    CONST robtarget Target_2550_2:=[[144.47,108.876,3],[0.69636424,0.122787804,0.122787804,-0.69636424],[-1,0,-1,1],[9E+09,9E+09,9E+09,9E+09,9E+09,9E+09]];
    CONST robtarget Target_2560_2:=[[144.866,108.509,3],[0.69636424,0.122787804,0.122787804,-0.69636424],[-1,0,-1,1],[9E+09,9E+09,9E+09,9E+09,9E+09,9E+09]];
    CONST robtarget Target_2570_2:=[[148.292,108.45,3],[0.69636424,0.122787804,0.122787804,-0.69636424],[-1,0,-1,1],[9E+09,9E+09,9E+09,9E+09,9E+09,9E+09]];
    CONST robtarget Target_2580_2:=[[149.079,109.372,3],[0.69636424,0.122787804,0.122787804,-0.69636424],[-1,0,-1,1],[9E+09,9E+09,9E+09,9E+09,9E+09,9E+09]];
    CONST robtarget Target_2590_2:=[[149.459,109.996,3],[0.69636424,0.122787804,0.122787804,-0.69636424],[-1,0,-1,1],[9E+09,9E+09,9E+09,9E+09,9E+09,9E+09]];
    CONST robtarget Target_2600_2:=[[149.804,110.629,3],[0.69636424,0.122787804,0.122787804,-0.69636424],[-1,0,-1,1],[9E+09,9E+09,9E+09,9E+09,9E+09,9E+09]];
    CONST robtarget Target_2610_2:=[[150.164,111.446,3],[0.69636424,0.122787804,0.122787804,-0.69636424],[-1,0,-1,1],[9E+09,9E+09,9E+09,9E+09,9E+09,9E+09]];
    CONST robtarget Target_2620_2:=[[150.582,112.397,3],[0.69636424,0.122787804,0.122787804,-0.69636424],[-1,0,-1,1],[9E+09,9E+09,9E+09,9E+09,9E+09,9E+09]];
    CONST robtarget Target_2630_2:=[[151.11,114.532,3],[0.69636424,0.122787804,0.122787804,-0.69636424],[-1,0,-1,1],[9E+09,9E+09,9E+09,9E+09,9E+09,9E+09]];
    CONST robtarget Target_2640_2:=[[151.258,118.351,3],[0.69636424,0.122787804,0.122787804,-0.69636424],[-1,0,-1,1],[9E+09,9E+09,9E+09,9E+09,9E+09,9E+09]];
    CONST robtarget Target_2650_2:=[[151.149,123.493,3],[0.69636424,0.122787804,0.122787804,-0.69636424],[-1,0,-1,1],[9E+09,9E+09,9E+09,9E+09,9E+09,9E+09]];
    CONST robtarget Target_2660_2:=[[150.509,124.998,3],[0.69636424,0.122787804,0.122787804,-0.69636424],[-1,0,-1,1],[9E+09,9E+09,9E+09,9E+09,9E+09,9E+09]];
    CONST robtarget Target_2670_2:=[[150.189,126.067,3],[0.69636424,0.122787804,0.122787804,-0.69636424],[-1,0,-1,1],[9E+09,9E+09,9E+09,9E+09,9E+09,9E+09]];
    CONST robtarget Target_2690_2:=[[149.435,127.495,3],[0.69636424,0.122787804,0.122787804,-0.69636424],[-1,0,-1,1],[9E+09,9E+09,9E+09,9E+09,9E+09,9E+09]];
    CONST robtarget Target_2700_2:=[[149.028,128.307,3],[0.69636424,0.122787804,0.122787804,-0.69636424],[-1,0,-1,1],[9E+09,9E+09,9E+09,9E+09,9E+09,9E+09]];
    CONST robtarget Target_2710_2:=[[148.353,128.811,3],[0.69636424,0.122787804,0.122787804,-0.69636424],[-1,0,-1,1],[9E+09,9E+09,9E+09,9E+09,9E+09,9E+09]];
    CONST robtarget Target_2720_2:=[[147.544,129.27,3],[0.69636424,0.122787804,0.122787804,-0.69636424],[-1,0,-1,1],[9E+09,9E+09,9E+09,9E+09,9E+09,9E+09]];
    CONST robtarget Target_2730_2:=[[146.677,129.693,3],[0.69636424,0.122787804,0.122787804,-0.69636424],[-1,0,-1,1],[9E+09,9E+09,9E+09,9E+09,9E+09,9E+09]];
    CONST robtarget Target_2740_2:=[[144.048,129.755,3],[0.69636424,0.122787804,0.122787804,-0.69636424],[-1,0,-1,1],[9E+09,9E+09,9E+09,9E+09,9E+09,9E+09]];
    CONST robtarget Target_2750_2:=[[141.627,127.645,3],[0.69636424,0.122787804,0.122787804,-0.69636424],[-1,0,-1,1],[9E+09,9E+09,9E+09,9E+09,9E+09,9E+09]];
    CONST robtarget Target_2760_2:=[[171.446,116.13,-27],[0.69636424,0.122787804,0.122787804,-0.69636424],[-1,0,-1,1],[9E+09,9E+09,9E+09,9E+09,9E+09,9E+09]];
    CONST robtarget Target_2770_2:=[[171.446,116.145,3],[0.69636424,0.122787804,0.122787804,-0.69636424],[-1,0,-1,1],[9E+09,9E+09,9E+09,9E+09,9E+09,9E+09]];
    CONST robtarget Target_2780_2:=[[171.382,110.454,3],[0.69636424,0.122787804,0.122787804,-0.69636424],[-1,0,-1,1],[9E+09,9E+09,9E+09,9E+09,9E+09,9E+09]];
    CONST robtarget Target_2790_2:=[[172.421,109.424,3],[0.69636424,0.122787804,0.122787804,-0.69636424],[-1,0,-1,1],[9E+09,9E+09,9E+09,9E+09,9E+09,9E+09]];
    CONST robtarget Target_2800_2:=[[173.527,108.448,3],[0.69636424,0.122787804,0.122787804,-0.69636424],[-1,0,-1,1],[9E+09,9E+09,9E+09,9E+09,9E+09,9E+09]];
    CONST robtarget Target_2810_2:=[[174.583,107.985,3],[0.69636424,0.122787804,0.122787804,-0.69636424],[-1,0,-1,1],[9E+09,9E+09,9E+09,9E+09,9E+09,9E+09]];
    CONST robtarget Target_2820_2:=[[175.225,107.505,3],[0.69636424,0.122787804,0.122787804,-0.69636424],[-1,0,-1,1],[9E+09,9E+09,9E+09,9E+09,9E+09,9E+09]];
    CONST robtarget Target_2830_2:=[[178.189,107.549,3],[0.69636424,0.122787804,0.122787804,-0.69636424],[-1,0,-1,1],[9E+09,9E+09,9E+09,9E+09,9E+09,9E+09]];
    CONST robtarget Target_2840_2:=[[178.951,108.484,3],[0.69636424,0.122787804,0.122787804,-0.69636424],[-1,0,-1,1],[9E+09,9E+09,9E+09,9E+09,9E+09,9E+09]];
    CONST robtarget Target_2850_2:=[[179.322,108.956,3],[0.69636424,0.122787804,0.122787804,-0.69636424],[-1,0,-1,1],[9E+09,9E+09,9E+09,9E+09,9E+09,9E+09]];
    CONST robtarget Target_2860_2:=[[179.662,109.677,3],[0.69636424,0.122787804,0.122787804,-0.69636424],[-1,0,-1,1],[9E+09,9E+09,9E+09,9E+09,9E+09,9E+09]];
    CONST robtarget Target_2870_2:=[[179.673,112.896,3],[0.69636424,0.122787804,0.122787804,-0.69636424],[-1,0,-1,1],[9E+09,9E+09,9E+09,9E+09,9E+09,9E+09]];
    CONST robtarget Target_2880_2:=[[178.94,113.73,3],[0.69636424,0.122787804,0.122787804,-0.69636424],[-1,0,-1,1],[9E+09,9E+09,9E+09,9E+09,9E+09,9E+09]];
    CONST robtarget Target_2890_2:=[[177.839,114.708,3],[0.69636424,0.122787804,0.122787804,-0.69636424],[-1,0,-1,1],[9E+09,9E+09,9E+09,9E+09,9E+09,9E+09]];
    CONST robtarget Target_2900_2:=[[175.361,115.711,3],[0.69636424,0.122787804,0.122787804,-0.69636424],[-1,0,-1,1],[9E+09,9E+09,9E+09,9E+09,9E+09,9E+09]];
    CONST robtarget Target_2910_2:=[[174.498,116.176,3],[0.69636424,0.122787804,0.122787804,-0.69636424],[-1,0,-1,1],[9E+09,9E+09,9E+09,9E+09,9E+09,9E+09]];
    CONST robtarget Target_2920_2:=[[207.225,82.129060431,2.819077862],[0.704416026,0.061628416,0.061628416,-0.704416026],[-1,0,-1,1],[9E+09,9E+09,9E+09,9E+09,9E+09,9E+09]];
    CONST robtarget Target_2920_up_2:=[[207.225,82.129060431,-27.180922138],[0.704416026,0.061628416,0.061628416,-0.704416026],[-1,0,-1,1],[9E+09,9E+09,9E+09,9E+09,9E+09,9E+09]];
    CONST robtarget Target_2930_2:=[[189.302,82.034060431,2.819077862],[0.704416026,0.061628416,0.061628416,-0.704416026],[-1,0,-1,1],[9E+09,9E+09,9E+09,9E+09,9E+09,9E+09]];
    CONST robtarget Target_2940_2:=[[172.295,56.628060431,2.819077862],[0.69636424,-0.122787804,-0.122787804,-0.69636424],[-1,0,-1,1],[9E+09,9E+09,9E+09,9E+09,9E+09,9E+09]];
    CONST robtarget Target_2950_2:=[[189.448,31.520060431,2.819077862],[0.704416026,0.061628416,0.061628416,-0.704416026],[-1,0,-1,1],[9E+09,9E+09,9E+09,9E+09,9E+09,9E+09]];
    CONST robtarget Target_2960_2:=[[207.063,31.366060431,2.819077862],[0.704416026,0.061628416,0.061628416,-0.704416026],[-1,0,-1,1],[9E+09,9E+09,9E+09,9E+09,9E+09,9E+09]];
    CONST robtarget Target_2970_2:=[[198.201,73.121060431,2.819077862],[0.704416026,0.061628416,0.061628416,-0.704416026],[-1,0,-1,1],[9E+09,9E+09,9E+09,9E+09,9E+09,9E+09]];
    CONST robtarget Target_2970_up_2:=[[198.201,73.121060431,-27.180922138],[0.704416026,0.061628416,0.061628416,-0.704416026],[-1,0,-1,1],[9E+09,9E+09,9E+09,9E+09,9E+09,9E+09]];
    CONST robtarget Target_2980_2:=[[189.482,72.946060431,2.819077862],[0.704416026,0.061628416,0.061628416,-0.704416026],[-1,0,-1,1],[9E+09,9E+09,9E+09,9E+09,9E+09,9E+09]];
    CONST robtarget Target_2990_2:=[[181.283,56.738060431,2.819077862],[0.69636424,-0.122787804,-0.122787804,-0.69636424],[-1,0,-1,1],[9E+09,9E+09,9E+09,9E+09,9E+09,9E+09]];
    CONST robtarget Target_3000_2:=[[189.826,40.515060431,2.819077862],[0.704416026,0.061628416,0.061628416,-0.704416026],[-1,0,-1,1],[9E+09,9E+09,9E+09,9E+09,9E+09,9E+09]];
    CONST robtarget Target_3010_2:=[[198.134,40.185060431,2.819077862],[0.704416026,0.061628416,0.061628416,-0.704416026],[-1,0,-1,1],[9E+09,9E+09,9E+09,9E+09,9E+09,9E+09]];
    CONST robtarget Target_3030_2_2:=[[168.856,62.045020144,-29.060307379],[0.704416026,0.061628416,0.061628416,-0.704416026],[-1,0,-1,1],[9E+09,9E+09,9E+09,9E+09,9E+09,9E+09]];
    CONST robtarget Target_3030_3:=[[168.856,62.729060431,2.819077862],[0.69636424,-0.122787804,-0.122787804,-0.69636424],[-1,0,-1,1],[9E+09,9E+09,9E+09,9E+09,9E+09,9E+09]];
    CONST robtarget Target_3040_2:=[[164.492,65.336020144,0.939692621],[0.704416026,0.061628416,0.061628416,-0.704416026],[-1,0,-1,1],[9E+09,9E+09,9E+09,9E+09,9E+09,9E+09]];
    CONST robtarget Target_3050_2:=[[159.783,67.041020144,0.939692621],[0.704416026,0.061628416,0.061628416,-0.704416026],[-1,0,-1,1],[9E+09,9E+09,9E+09,9E+09,9E+09,9E+09]];
    CONST robtarget Target_3060_2:=[[154.529,67.248020144,0.939692621],[0.704416026,0.061628416,0.061628416,-0.704416026],[-1,0,-1,1],[9E+09,9E+09,9E+09,9E+09,9E+09,9E+09]];
    CONST robtarget Target_3070_2:=[[149.168,63.265020144,0.939692621],[0.704416026,0.061628416,0.061628416,-0.704416026],[-1,0,-1,1],[9E+09,9E+09,9E+09,9E+09,9E+09,9E+09]];
    CONST robtarget Target_3080_2:=[[146.594,56.470020144,0.939692621],[0.704416026,0.061628416,0.061628416,-0.704416026],[-1,0,-1,1],[9E+09,9E+09,9E+09,9E+09,9E+09,9E+09]];
    CONST robtarget Target_3090_2:=[[146.435,30.622020144,0.939692621],[0.704416026,0.061628416,0.061628416,-0.704416026],[-1,0,-1,1],[9E+09,9E+09,9E+09,9E+09,9E+09,9E+09]];
    CONST robtarget Target_3100_2:=[[151.326,30.602020144,0.939692621],[0.704416026,0.061628416,0.061628416,-0.704416026],[-1,0,-1,1],[9E+09,9E+09,9E+09,9E+09,9E+09,9E+09]];
    CONST robtarget Target_3110_2:=[[153.44,34.909020144,0.939692621],[0.704416026,0.061628416,0.061628416,-0.704416026],[-1,0,-1,1],[9E+09,9E+09,9E+09,9E+09,9E+09,9E+09]];
    CONST robtarget Target_3120_2:=[[156.57,31.843020144,0.939692621],[0.704416026,0.061628416,0.061628416,-0.704416026],[-1,0,-1,1],[9E+09,9E+09,9E+09,9E+09,9E+09,9E+09]];
    CONST robtarget Target_3130_2:=[[160.302,30.191020144,0.939692621],[0.704416026,0.061628416,0.061628416,-0.704416026],[-1,0,-1,1],[9E+09,9E+09,9E+09,9E+09,9E+09,9E+09]];
    CONST robtarget Target_3140_2:=[[163.825,30.168020144,0.939692621],[0.704416026,0.061628416,0.061628416,-0.704416026],[-1,0,-1,1],[9E+09,9E+09,9E+09,9E+09,9E+09,9E+09]];
    CONST robtarget Target_3150_2:=[[167.12,31.969020144,0.939692621],[0.704416026,0.061628416,0.061628416,-0.704416026],[-1,0,-1,1],[9E+09,9E+09,9E+09,9E+09,9E+09,9E+09]];
    CONST robtarget Target_3160_2:=[[169.87,36.987020144,0.939692621],[0.704416026,0.061628416,0.061628416,-0.704416026],[-1,0,-1,1],[9E+09,9E+09,9E+09,9E+09,9E+09,9E+09]];
    CONST robtarget Target_3170_2:=[[170.005,41.186020144,0.939692621],[0.704416026,0.061628416,0.061628416,-0.704416026],[-1,0,-1,1],[9E+09,9E+09,9E+09,9E+09,9E+09,9E+09]];
    CONST robtarget Target_3180_2:=[[166.518,48.057020144,0.939692621],[0.704416026,0.061628416,0.061628416,-0.704416026],[-1,0,-1,1],[9E+09,9E+09,9E+09,9E+09,9E+09,9E+09]];
    CONST robtarget Target_3190_2:=[[159.562,51.317020144,0.939692621],[0.704416026,0.061628416,0.061628416,-0.704416026],[-1,0,-1,1],[9E+09,9E+09,9E+09,9E+09,9E+09,9E+09]];
    CONST robtarget Target_3200_2:=[[154.356,51.836020144,0.939692621],[0.704416026,0.061628416,0.061628416,-0.704416026],[-1,0,-1,1],[9E+09,9E+09,9E+09,9E+09,9E+09,9E+09]];
    CONST robtarget Target_3210_2:=[[154.402,56.254020144,0.939692621],[0.704416026,0.061628416,0.061628416,-0.704416026],[-1,0,-1,1],[9E+09,9E+09,9E+09,9E+09,9E+09,9E+09]];
    CONST robtarget Target_3220_2:=[[156.646,59.021020144,0.939692621],[0.704416026,0.061628416,0.061628416,-0.704416026],[-1,0,-1,1],[9E+09,9E+09,9E+09,9E+09,9E+09,9E+09]];
    CONST robtarget Target_3230_2:=[[159.999,59.059020144,0.939692621],[0.704416026,0.061628416,0.061628416,-0.704416026],[-1,0,-1,1],[9E+09,9E+09,9E+09,9E+09,9E+09,9E+09]];
    CONST robtarget Target_3240_2:=[[163.724,56.946020144,0.939692621],[0.704416026,0.061628416,0.061628416,-0.704416026],[-1,0,-1,1],[9E+09,9E+09,9E+09,9E+09,9E+09,9E+09]];
    CONST robtarget Target_3250_2:=[[166.309,56.964020144,0.939692621],[0.704416026,0.061628416,0.061628416,-0.704416026],[-1,0,-1,1],[9E+09,9E+09,9E+09,9E+09,9E+09,9E+09]];
    CONST robtarget Target_3260_2_2:=[[154.254,45.587020144,-29.060307379],[0.704416026,0.061628416,0.061628416,-0.704416026],[-1,0,-1,1],[9E+09,9E+09,9E+09,9E+09,9E+09,9E+09]];
    CONST robtarget Target_3260_3:=[[154.254,45.587020144,0.939692621],[0.69636424,-0.122787804,-0.122787804,-0.69636424],[-1,0,-1,1],[9E+09,9E+09,9E+09,9E+09,9E+09,9E+09]];
    CONST robtarget Target_3270_2:=[[154.243,40.170020144,0.939692621],[0.704416026,0.061628416,0.061628416,-0.704416026],[-1,0,-1,1],[9E+09,9E+09,9E+09,9E+09,9E+09,9E+09]];
    CONST robtarget Target_3280_2:=[[155.887,38.274020144,0.939692621],[0.704416026,0.061628416,0.061628416,-0.704416026],[-1,0,-1,1],[9E+09,9E+09,9E+09,9E+09,9E+09,9E+09]];
    CONST robtarget Target_3290_2:=[[157.675,37.336020144,0.939692621],[0.704416026,0.061628416,0.061628416,-0.704416026],[-1,0,-1,1],[9E+09,9E+09,9E+09,9E+09,9E+09,9E+09]];
    CONST robtarget Target_3300_2:=[[160.603,37.207020144,0.939692621],[0.704416026,0.061628416,0.061628416,-0.704416026],[-1,0,-1,1],[9E+09,9E+09,9E+09,9E+09,9E+09,9E+09]];
    CONST robtarget Target_3310_2:=[[162.533,39.193020144,0.939692621],[0.704416026,0.061628416,0.061628416,-0.704416026],[-1,0,-1,1],[9E+09,9E+09,9E+09,9E+09,9E+09,9E+09]];
    CONST robtarget Target_3320_2:=[[162.426,41.941020144,0.939692621],[0.704416026,0.061628416,0.061628416,-0.704416026],[-1,0,-1,1],[9E+09,9E+09,9E+09,9E+09,9E+09,9E+09]];
    CONST robtarget Target_3330_2:=[[160.229,44.430020144,0.939692621],[0.704416026,0.061628416,0.061628416,-0.704416026],[-1,0,-1,1],[9E+09,9E+09,9E+09,9E+09,9E+09,9E+09]];
    CONST robtarget Target_3340_2:=[[157.734,45.576020144,0.939692621],[0.704416026,0.061628416,0.061628416,-0.704416026],[-1,0,-1,1],[9E+09,9E+09,9E+09,9E+09,9E+09,9E+09]];
    CONST robtarget Target_3350_2_2:=[[144.461,67.032020144,-29.060307379],[0.704416026,0.061628416,0.061628416,-0.704416026],[-1,0,-1,1],[9E+09,9E+09,9E+09,9E+09,9E+09,9E+09]];
    CONST robtarget Target_3350_3:=[[144.461,67.032020144,0.939692621],[0.69636424,-0.122787804,-0.122787804,-0.69636424],[-1,0,-1,1],[9E+09,9E+09,9E+09,9E+09,9E+09,9E+09]];
    CONST robtarget Target_3360_2:=[[136.399,66.775020144,0.939692621],[0.704416026,0.061628416,0.061628416,-0.704416026],[-1,0,-1,1],[9E+09,9E+09,9E+09,9E+09,9E+09,9E+09]];
    CONST robtarget Target_3370_2:=[[130.223,41.577020144,0.939692621],[0.704416026,0.061628416,0.061628416,-0.704416026],[-1,0,-1,1],[9E+09,9E+09,9E+09,9E+09,9E+09,9E+09]];
    CONST robtarget Target_3380_2:=[[123.937,66.551020144,0.939692621],[0.704416026,0.061628416,0.061628416,-0.704416026],[-1,0,-1,1],[9E+09,9E+09,9E+09,9E+09,9E+09,9E+09]];
    CONST robtarget Target_3390_2:=[[115.96,66.627020144,0.939692621],[0.704416026,0.061628416,0.061628416,-0.704416026],[-1,0,-1,1],[9E+09,9E+09,9E+09,9E+09,9E+09,9E+09]];
    CONST robtarget Target_3400_2:=[[126.475,30.638020144,0.939692621],[0.704416026,0.061628416,0.061628416,-0.704416026],[-1,0,-1,1],[9E+09,9E+09,9E+09,9E+09,9E+09,9E+09]];
    CONST robtarget Target_3410_2:=[[133.864,30.673020144,0.939692621],[0.704416026,0.061628416,0.061628416,-0.704416026],[-1,0,-1,1],[9E+09,9E+09,9E+09,9E+09,9E+09,9E+09]];
    CONST robtarget Target_3420_2_2:=[[112.825,66.820020144,-29.060307379],[0.704416026,0.061628416,0.061628416,-0.704416026],[-1,0,-1,1],[9E+09,9E+09,9E+09,9E+09,9E+09,9E+09]];
    CONST robtarget Target_3420_3:=[[112.825,66.820020144,0.939692621],[0.69636424,-0.122787804,-0.122787804,-0.69636424],[-1,0,-1,1],[9E+09,9E+09,9E+09,9E+09,9E+09,9E+09]];
    CONST robtarget Target_3430_2:=[[104.746,66.822020144,0.939692621],[0.704416026,0.061628416,0.061628416,-0.704416026],[-1,0,-1,1],[9E+09,9E+09,9E+09,9E+09,9E+09,9E+09]];
    CONST robtarget Target_3440_2:=[[104.632,30.482020144,0.939692621],[0.704416026,0.061628416,0.061628416,-0.704416026],[-1,0,-1,1],[9E+09,9E+09,9E+09,9E+09,9E+09,9E+09]];
    CONST robtarget Target_3450_2:=[[112.782,30.740020144,0.939692621],[0.704416026,0.061628416,0.061628416,-0.704416026],[-1,0,-1,1],[9E+09,9E+09,9E+09,9E+09,9E+09,9E+09]];
    CONST robtarget Target_3460_2_2:=[[107.732,82.799020144,-29.060307379],[0.704416026,0.061628416,0.061628416,-0.704416026],[-1,0,-1,1],[9E+09,9E+09,9E+09,9E+09,9E+09,9E+09]];
    CONST robtarget Target_3460_3:=[[107.732,82.799020144,0.939692621],[0.69636424,-0.122787804,-0.122787804,-0.69636424],[-1,0,-1,1],[9E+09,9E+09,9E+09,9E+09,9E+09,9E+09]];
    CONST robtarget Target_3470_2:=[[103.914,76.496020144,0.939692621],[0.704416026,0.061628416,0.061628416,-0.704416026],[-1,0,-1,1],[9E+09,9E+09,9E+09,9E+09,9E+09,9E+09]];
    CONST robtarget Target_3480_2:=[[107.812,70.304020144,0.939692621],[0.704416026,0.061628416,0.061628416,-0.704416026],[-1,0,-1,1],[9E+09,9E+09,9E+09,9E+09,9E+09,9E+09]];
    CONST robtarget Target_3490_2:=[[110.105,70.397020144,0.939692621],[0.704416026,0.061628416,0.061628416,-0.704416026],[-1,0,-1,1],[9E+09,9E+09,9E+09,9E+09,9E+09,9E+09]];
    CONST robtarget Target_3500_2:=[[113.61,76.180020144,0.939692621],[0.704416026,0.061628416,0.061628416,-0.704416026],[-1,0,-1,1],[9E+09,9E+09,9E+09,9E+09,9E+09,9E+09]];
    CONST robtarget Target_3510_2:=[[110.04,82.825020144,0.939692621],[0.704416026,0.061628416,0.061628416,-0.704416026],[-1,0,-1,1],[9E+09,9E+09,9E+09,9E+09,9E+09,9E+09]];
    CONST robtarget Target_3520_2_2:=[[82.277,82.761020144,-29.060307379],[0.704416026,0.061628416,0.061628416,-0.704416026],[-1,0,-1,1],[9E+09,9E+09,9E+09,9E+09,9E+09,9E+09]];
    CONST robtarget Target_3520_3:=[[82.277,82.761020144,0.939692621],[0.69636424,-0.122787804,-0.122787804,-0.69636424],[-1,0,-1,1],[9E+09,9E+09,9E+09,9E+09,9E+09,9E+09]];
    CONST robtarget Target_3530_2:=[[74.455,82.673020144,0.939692621],[0.704416026,0.061628416,0.061628416,-0.704416026],[-1,0,-1,1],[9E+09,9E+09,9E+09,9E+09,9E+09,9E+09]];
    CONST robtarget Target_3540_2:=[[74.428,30.709020144,0.939692621],[0.704416026,0.061628416,0.061628416,-0.704416026],[-1,0,-1,1],[9E+09,9E+09,9E+09,9E+09,9E+09,9E+09]];
    CONST robtarget Target_3550_2:=[[80.004,30.702020144,0.939692621],[0.704416026,0.061628416,0.061628416,-0.704416026],[-1,0,-1,1],[9E+09,9E+09,9E+09,9E+09,9E+09,9E+09]];
    CONST robtarget Target_3560_2:=[[82.07,35.013020144,0.939692621],[0.704416026,0.061628416,0.061628416,-0.704416026],[-1,0,-1,1],[9E+09,9E+09,9E+09,9E+09,9E+09,9E+09]];
    CONST robtarget Target_3570_2:=[[84.954,31.898020144,0.939692621],[0.704416026,0.061628416,0.061628416,-0.704416026],[-1,0,-1,1],[9E+09,9E+09,9E+09,9E+09,9E+09,9E+09]];
    CONST robtarget Target_3580_2:=[[88.431,30.331020144,0.939692621],[0.704416026,0.061628416,0.061628416,-0.704416026],[-1,0,-1,1],[9E+09,9E+09,9E+09,9E+09,9E+09,9E+09]];
    CONST robtarget Target_3590_2:=[[92.072,30.216020144,0.939692621],[0.704416026,0.061628416,0.061628416,-0.704416026],[-1,0,-1,1],[9E+09,9E+09,9E+09,9E+09,9E+09,9E+09]];
    CONST robtarget Target_3600_2:=[[97.435,34.873020144,0.939692621],[0.704416026,0.061628416,0.061628416,-0.704416026],[-1,0,-1,1],[9E+09,9E+09,9E+09,9E+09,9E+09,9E+09]];
    CONST robtarget Target_3610_2:=[[99.865,42.963020144,0.939692621],[0.704416026,0.061628416,0.061628416,-0.704416026],[-1,0,-1,1],[9E+09,9E+09,9E+09,9E+09,9E+09,9E+09]];
    CONST robtarget Target_3620_2:=[[100.165,49.389020144,0.939692621],[0.704416026,0.061628416,0.061628416,-0.704416026],[-1,0,-1,1],[9E+09,9E+09,9E+09,9E+09,9E+09,9E+09]];
    CONST robtarget Target_3630_2:=[[97.664,60.583020144,0.939692621],[0.704416026,0.061628416,0.061628416,-0.704416026],[-1,0,-1,1],[9E+09,9E+09,9E+09,9E+09,9E+09,9E+09]];
    CONST robtarget Target_3640_2:=[[90.704,67.178020144,0.939692621],[0.704416026,0.061628416,0.061628416,-0.704416026],[-1,0,-1,1],[9E+09,9E+09,9E+09,9E+09,9E+09,9E+09]];
    CONST robtarget Target_3650_2:=[[86.592,67.289020144,0.939692621],[0.704416026,0.061628416,0.061628416,-0.704416026],[-1,0,-1,1],[9E+09,9E+09,9E+09,9E+09,9E+09,9E+09]];
    CONST robtarget Target_3660_2:=[[82.282,64.136020144,0.939692621],[0.704416026,0.061628416,0.061628416,-0.704416026],[-1,0,-1,1],[9E+09,9E+09,9E+09,9E+09,9E+09,9E+09]];
    CONST robtarget Target_3670_2_2:=[[82.253,56.509020144,-29.060307379],[0.704416026,0.061628416,0.061628416,-0.704416026],[-1,0,-1,1],[9E+09,9E+09,9E+09,9E+09,9E+09,9E+09]];
    CONST robtarget Target_3670_3:=[[82.253,56.509020144,0.939692621],[0.69636424,-0.122787804,-0.122787804,-0.69636424],[-1,0,-1,1],[9E+09,9E+09,9E+09,9E+09,9E+09,9E+09]];
    CONST robtarget Target_3680_2:=[[82.272,41.520020144,0.939692621],[0.704416026,0.061628416,0.061628416,-0.704416026],[-1,0,-1,1],[9E+09,9E+09,9E+09,9E+09,9E+09,9E+09]];
    CONST robtarget Target_3690_2:=[[85.391,38.217020144,0.939692621],[0.704416026,0.061628416,0.061628416,-0.704416026],[-1,0,-1,1],[9E+09,9E+09,9E+09,9E+09,9E+09,9E+09]];
    CONST robtarget Target_3700_2:=[[88.811,38.071020144,0.939692621],[0.704416026,0.061628416,0.061628416,-0.704416026],[-1,0,-1,1],[9E+09,9E+09,9E+09,9E+09,9E+09,9E+09]];
    CONST robtarget Target_3710_2:=[[91.889,43.979020144,0.939692621],[0.704416026,0.061628416,0.061628416,-0.704416026],[-1,0,-1,1],[9E+09,9E+09,9E+09,9E+09,9E+09,9E+09]];
    CONST robtarget Target_3720_2:=[[92.083,51.104020144,0.939692621],[0.704416026,0.061628416,0.061628416,-0.704416026],[-1,0,-1,1],[9E+09,9E+09,9E+09,9E+09,9E+09,9E+09]];
    CONST robtarget Target_3730_2:=[[89.43,58.065020144,0.939692621],[0.704416026,0.061628416,0.061628416,-0.704416026],[-1,0,-1,1],[9E+09,9E+09,9E+09,9E+09,9E+09,9E+09]];
    CONST robtarget Target_3740_2:=[[85.526,58.965020144,0.939692621],[0.704416026,0.061628416,0.061628416,-0.704416026],[-1,0,-1,1],[9E+09,9E+09,9E+09,9E+09,9E+09,9E+09]];
    CONST robtarget Target_3750_2_2:=[[64.524,146.437020144,-29.060307379],[0.704416026,0.061628416,0.061628416,-0.704416026],[-1,0,-1,1],[9E+09,9E+09,9E+09,9E+09,9E+09,9E+09]];
    CONST robtarget Target_3750_3:=[[64.524,146.437020144,0.939692621],[0.69636424,-0.122787804,-0.122787804,-0.69636424],[-1,0,-1,1],[9E+09,9E+09,9E+09,9E+09,9E+09,9E+09]];
    CONST robtarget Target_3760_2:=[[55.549,133.666020144,0.939692621],[0.704416026,0.061628416,0.061628416,-0.704416026],[-1,0,-1,1],[9E+09,9E+09,9E+09,9E+09,9E+09,9E+09]];
    CONST robtarget Target_3770_2:=[[47.044,128.487020144,0.939692621],[0.704416026,0.061628416,0.061628416,-0.704416026],[-1,0,-1,1],[9E+09,9E+09,9E+09,9E+09,9E+09,9E+09]];
    CONST robtarget Target_3780_2:=[[37.688,111.228020144,0.939692621],[0.704416026,0.061628416,0.061628416,-0.704416026],[-1,0,-1,1],[9E+09,9E+09,9E+09,9E+09,9E+09,9E+09]];
    CONST robtarget Target_3790_2:=[[41.259,123.994020144,0.939692621],[0.704416026,0.061628416,0.061628416,-0.704416026],[-1,0,-1,1],[9E+09,9E+09,9E+09,9E+09,9E+09,9E+09]];
    CONST robtarget Target_3800_2:=[[26.923,126.980020144,0.939692621],[0.704416026,0.061628416,0.061628416,-0.704416026],[-1,0,-1,1],[9E+09,9E+09,9E+09,9E+09,9E+09,9E+09]];
    CONST robtarget Target_3810_2:=[[26.91,85.429020144,0.939692621],[0.704416026,0.061628416,0.061628416,-0.704416026],[-1,0,-1,1],[9E+09,9E+09,9E+09,9E+09,9E+09,9E+09]];
    CONST robtarget Target_3820_2:=[[31.003,81.597020144,0.939692621],[0.704416026,0.061628416,0.061628416,-0.704416026],[-1,0,-1,1],[9E+09,9E+09,9E+09,9E+09,9E+09,9E+09]];
    CONST robtarget Target_3830_2:=[[35.653,89.236020144,0.939692621],[0.704416026,0.061628416,0.061628416,-0.704416026],[-1,0,-1,1],[9E+09,9E+09,9E+09,9E+09,9E+09,9E+09]];
    CONST robtarget Target_3840_2:=[[41.161,97.045020144,0.939692621],[0.704416026,0.061628416,0.061628416,-0.704416026],[-1,0,-1,1],[9E+09,9E+09,9E+09,9E+09,9E+09,9E+09]];
    CONST robtarget Target_3850_2:=[[45.695,102.026020144,0.939692621],[0.704416026,0.061628416,0.061628416,-0.704416026],[-1,0,-1,1],[9E+09,9E+09,9E+09,9E+09,9E+09,9E+09]];
    CONST robtarget Target_3860_2:=[[52.946,106.880020144,0.939692621],[0.704416026,0.061628416,0.061628416,-0.704416026],[-1,0,-1,1],[9E+09,9E+09,9E+09,9E+09,9E+09,9E+09]];
    CONST robtarget Target_3870_2:=[[62.408,123.824020144,0.939692621],[0.704416026,0.061628416,0.061628416,-0.704416026],[-1,0,-1,1],[9E+09,9E+09,9E+09,9E+09,9E+09,9E+09]];
    CONST robtarget Target_3880_2:=[[52.276,112.163020144,0.939692621],[0.704416026,0.061628416,0.061628416,-0.704416026],[-1,0,-1,1],[9E+09,9E+09,9E+09,9E+09,9E+09,9E+09]];
    CONST robtarget Target_3890_2:=[[59.313,122.581020144,0.939692621],[0.704416026,0.061628416,0.061628416,-0.704416026],[-1,0,-1,1],[9E+09,9E+09,9E+09,9E+09,9E+09,9E+09]];
    CONST robtarget Target_3900_2:=[[63.763,135.404020144,0.939692621],[0.704416026,0.061628416,0.061628416,-0.704416026],[-1,0,-1,1],[9E+09,9E+09,9E+09,9E+09,9E+09,9E+09]];
    CONST robtarget Target_3910_2_2:=[[27.611,83.068020144,-29.060307379],[0.704416026,0.061628416,0.061628416,-0.704416026],[-1,0,-1,1],[9E+09,9E+09,9E+09,9E+09,9E+09,9E+09]];
    CONST robtarget Target_3910_3:=[[27.611,83.068020144,0.939692621],[0.69636424,-0.122787804,-0.122787804,-0.69636424],[-1,0,-1,1],[9E+09,9E+09,9E+09,9E+09,9E+09,9E+09]];
    CONST robtarget Target_3920_2:=[[24.514,80.149020144,0.939692621],[0.704416026,0.061628416,0.061628416,-0.704416026],[-1,0,-1,1],[9E+09,9E+09,9E+09,9E+09,9E+09,9E+09]];
    CONST robtarget Target_3930_2:=[[24.493,70.759020144,0.939692621],[0.704416026,0.061628416,0.061628416,-0.704416026],[-1,0,-1,1],[9E+09,9E+09,9E+09,9E+09,9E+09,9E+09]];
    CONST robtarget Target_3940_2:=[[26.846,61.477020144,0.939692621],[0.704416026,0.061628416,0.061628416,-0.704416026],[-1,0,-1,1],[9E+09,9E+09,9E+09,9E+09,9E+09,9E+09]];
    CONST robtarget Target_3950_2:=[[29.828,69.272020144,0.939692621],[0.704416026,0.061628416,0.061628416,-0.704416026],[-1,0,-1,1],[9E+09,9E+09,9E+09,9E+09,9E+09,9E+09]];
    CONST robtarget Target_3960_2:=[[30.012,78.359020144,0.939692621],[0.704416026,0.061628416,0.061628416,-0.704416026],[-1,0,-1,1],[9E+09,9E+09,9E+09,9E+09,9E+09,9E+09]];
    CONST robtarget Target_3970_2_2:=[[44.273,96.711020144,-29.060307379],[0.704416026,0.061628416,0.061628416,-0.704416026],[-1,0,-1,1],[9E+09,9E+09,9E+09,9E+09,9E+09,9E+09]];
    CONST robtarget Target_3970_3:=[[44.273,96.711020144,0.939692621],[0.69636424,-0.122787804,-0.122787804,-0.69636424],[-1,0,-1,1],[9E+09,9E+09,9E+09,9E+09,9E+09,9E+09]];
    CONST robtarget Target_3980_2:=[[43.933,86.227020144,0.939692621],[0.704416026,0.061628416,0.061628416,-0.704416026],[-1,0,-1,1],[9E+09,9E+09,9E+09,9E+09,9E+09,9E+09]];
    CONST robtarget Target_3990_2:=[[39.768,82.418020144,0.939692621],[0.704416026,0.061628416,0.061628416,-0.704416026],[-1,0,-1,1],[9E+09,9E+09,9E+09,9E+09,9E+09,9E+09]];
    CONST robtarget Target_4000_2:=[[34.596,82.452020144,0.939692621],[0.704416026,0.061628416,0.061628416,-0.704416026],[-1,0,-1,1],[9E+09,9E+09,9E+09,9E+09,9E+09,9E+09]];
    CONST robtarget Target_4010_2_2:=[[26.792,57.803020144,-29.060307379],[0.704416026,0.061628416,0.061628416,-0.704416026],[-1,0,-1,1],[9E+09,9E+09,9E+09,9E+09,9E+09,9E+09]];
    CONST robtarget Target_4010_3:=[[26.792,57.803020144,0.939692621],[0.69636424,-0.122787804,-0.122787804,-0.69636424],[-1,0,-1,1],[9E+09,9E+09,9E+09,9E+09,9E+09,9E+09]];
    CONST robtarget Target_4020_2:=[[45.072,60.926020144,0.939692621],[0.704416026,0.061628416,0.061628416,-0.704416026],[-1,0,-1,1],[9E+09,9E+09,9E+09,9E+09,9E+09,9E+09]];
    CONST robtarget Target_4030_2:=[[61.878,52.724020144,0.939692621],[0.704416026,0.061628416,0.061628416,-0.704416026],[-1,0,-1,1],[9E+09,9E+09,9E+09,9E+09,9E+09,9E+09]];
    CONST robtarget Target_4040_2:=[[59.898,63.620020144,0.939692621],[0.704416026,0.061628416,0.061628416,-0.704416026],[-1,0,-1,1],[9E+09,9E+09,9E+09,9E+09,9E+09,9E+09]];
    CONST robtarget Target_4050_2:=[[56.445,72.459020144,0.939692621],[0.704416026,0.061628416,0.061628416,-0.704416026],[-1,0,-1,1],[9E+09,9E+09,9E+09,9E+09,9E+09,9E+09]];
    CONST robtarget Target_4060_2:=[[58.835,86.000020144,0.939692621],[0.704416026,0.061628416,0.061628416,-0.704416026],[-1,0,-1,1],[9E+09,9E+09,9E+09,9E+09,9E+09,9E+09]];
    CONST robtarget Target_4070_2:=[[54.916,107.364020144,0.939692621],[0.704416026,0.061628416,0.061628416,-0.704416026],[-1,0,-1,1],[9E+09,9E+09,9E+09,9E+09,9E+09,9E+09]];
    CONST robtarget Target_4080_2:=[[49.508,100.246020144,0.939692621],[0.704416026,0.061628416,0.061628416,-0.704416026],[-1,0,-1,1],[9E+09,9E+09,9E+09,9E+09,9E+09,9E+09]];
    CONST robtarget Target_4090_2:=[[52.038,93.753020144,0.939692621],[0.704416026,0.061628416,0.061628416,-0.704416026],[-1,0,-1,1],[9E+09,9E+09,9E+09,9E+09,9E+09,9E+09]];
    CONST robtarget Target_4100_2:=[[52.392,84.414020144,0.939692621],[0.704416026,0.061628416,0.061628416,-0.704416026],[-1,0,-1,1],[9E+09,9E+09,9E+09,9E+09,9E+09,9E+09]];
    CONST robtarget Target_4110_2:=[[48.592,78.019020144,0.939692621],[0.704416026,0.061628416,0.061628416,-0.704416026],[-1,0,-1,1],[9E+09,9E+09,9E+09,9E+09,9E+09,9E+09]];
    CONST robtarget Target_4120_2:=[[44.019,73.976020144,0.939692621],[0.704416026,0.061628416,0.061628416,-0.704416026],[-1,0,-1,1],[9E+09,9E+09,9E+09,9E+09,9E+09,9E+09]];
    CONST robtarget Target_4130_2:=[[36.693,67.321020144,0.939692621],[0.704416026,0.061628416,0.061628416,-0.704416026],[-1,0,-1,1],[9E+09,9E+09,9E+09,9E+09,9E+09,9E+09]];



    PROC main()
        TPErase;
        TPWrite "Iniciando Ciclo";
        !Aqui  se reinicia todas las entradas y salidad a usar.
        Reset Conveyor_INV;
        Reset DO_01;
        Reset DO_02;
        GoHome;
        TPWrite "Porfavor presione Bot n1 para iniciar Rutina de decoracion ";
        TPWrite "Tambien, puede presionar Bot n2 para iniciar Rutina de Matenimiento ";

   WHILE TRUE DO
            IF DI_01 = 1 AND DI_02 = 0 THEN  !verificar que solo se presiono un bot n
                TPWrite "Comenzando avance de la banda";
                Set Conveyor_INV;
                WaitTime 8.7;  !cambiar este para modificar tiempo de espera entre encendido y apagado 10.2 simulaci n, 4 en real
                Reset Conveyor_INV;
                TPWrite "Banda transportadora detenida";
                TPWrite "Iniciando Decoraci n del pastel";
                Set DO_01; ! bombillo que avisa del proceso de decoraci n
                MoveAbsJ RomperSingular, v1000, z1, Soporte_final;
                Path_40;
                Path_10; ! Primero Ariadna
                TPWrite "Decoraci n ------> 34%";
                Path_20;
                TPWrite "Decoraci n ------> 67%";
                Path_30;
                TPWrite "Decoraci n ------> 100%";
                GoHome;
                WaitTime 2; !verificar este Gohome que hace.
                TPWrite "Comenzando avance de la banda";
                Set Conveyor_INV;
                WaitTime 3; ! si la caja se cae es por esto en simulaci n 3, 0.2 en real
                Reset Conveyor_INV;
                TPWrite "Banda transportadora detenida";


            ELSEIF DI_01 = 0 AND DI_02=1 THEN
                TPWrite "Rutina de Mantenimiento empezando";
                Reset DO_01; ! apagando indicador de rutina de decoraci n
                Set DO_02; ! indicador de la rutina de mantenimiento
                GoHome;
                MoveAbsJ cambio_Tool, v300, z5, Soporte_final;
                TPWrite "CUIDADO OPERARIO CERCA AL ROBOT";
                TPWrite "Presione Boton1 y Boton2 al tiempo, para continuar";
                WaitUntil DI_01=1 AND DI_02=1;
                TPWrite "Continuando Programa...";
                WaitTime 6; ! tiempo de espera para asegurarse que el operario salio.
                MoveAbsJ HOME_Origen, v300, fine, Soporte_final;
                Reset DO_02;
            ELSEIF DI_01 = 0 AND DI_02=0 THEN
                TPWrite "Esperando Instrucciones";
                ! aqui iba un Waittime pero no pienso que sea neccesario
            ENDIF
             ! revisar si es necesario otro estado
        ENDWHILE


    ENDPROC

       PROC GoHome()
        CONST num tolerancia := 0.2;
        VAR jointtarget jt;
        jt := CJointT(); ! posici n actual del robot
        IF  Abs(jt.robax.rax_1) < tolerancia AND
            Abs(jt.robax.rax_2) < tolerancia AND
            Abs(jt.robax.rax_3) < tolerancia AND
            Abs(jt.robax.rax_4) < tolerancia AND
            Abs(jt.robax.rax_5) < tolerancia AND
            Abs(jt.robax.rax_6) < tolerancia THEN
            TPWrite "Robot en home articular en 0 ";
        ELSE
            TPWrite "Yendo a Home";

            MoveAbsJ HOME_Origen, v100, fine, Soporte_final;
            TPWrite "Robot en Home";
        ENDIF
    ENDPROC

  PROC Path_10()
        MoveJ Target_minihome,v100,z5,Soporte_final\WObj:=ADwob;
        MoveJ Target_200,v100,z5,Soporte_final\WObj:=ADwob;
        MoveL Target_210,v100,z5,Soporte_final\WObj:=ADwob;
        MoveL Target_220,v100,z5,Soporte_final\WObj:=ADwob;
        MoveL Target_230,v100,z5,Soporte_final\WObj:=ADwob;
        MoveL Target_240,v100,z5,Soporte_final\WObj:=ADwob;
        MoveL Target_250,v100,z5,Soporte_final\WObj:=ADwob;
        MoveL Target_260,v100,z5,Soporte_final\WObj:=ADwob;
        MoveL Target_270,v100,z5,Soporte_final\WObj:=ADwob;
        MoveL Target_280,v100,z5,Soporte_final\WObj:=ADwob;
        MoveL Target_210,v100,z5,Soporte_final\WObj:=ADwob;
        MoveL Target_200,v100,z5,Soporte_final\WObj:=ADwob;
        MoveL Target_290,v100,z5,Soporte_final\WObj:=ADwob;
        MoveL Target_300,v100,z5,Soporte_final\WObj:=ADwob;
        MoveL Target_310,v100,z5,Soporte_final\WObj:=ADwob;
        MoveL Target_320,v100,z5,Soporte_final\WObj:=ADwob;
        MoveL Target_300,v100,z5,Soporte_final\WObj:=ADwob;
        MoveL Target_290,v100,z5,Soporte_final\WObj:=ADwob;
        MoveL Target_330,v100,z5,Soporte_final\WObj:=ADwob;
        MoveL Target_340,v100,z5,Soporte_final\WObj:=ADwob;
        MoveL Target_350,v100,z5,Soporte_final\WObj:=ADwob;
        MoveL Target_360,v100,z5,Soporte_final\WObj:=ADwob;
        MoveL Target_370,v100,z5,Soporte_final\WObj:=ADwob;
        MoveL Target_380,v100,z5,Soporte_final\WObj:=ADwob;
        MoveL Target_390,v100,z5,Soporte_final\WObj:=ADwob;
        MoveL Target_400,v100,z5,Soporte_final\WObj:=ADwob;
        MoveL Target_410,v100,z5,Soporte_final\WObj:=ADwob;
        MoveL Target_420,v100,z5,Soporte_final\WObj:=ADwob;
        MoveL Target_430,v100,z5,Soporte_final\WObj:=ADwob;
        MoveL Target_440,v100,z5,Soporte_final\WObj:=ADwob;
        MoveL Target_340,v100,z5,Soporte_final\WObj:=ADwob;
        MoveL Target_330,v100,z5,Soporte_final\WObj:=ADwob;
        MoveL Target_450,v100,z5,Soporte_final\WObj:=ADwob;
        MoveL Target_460,v100,z5,Soporte_final\WObj:=ADwob;
        MoveL Target_470,v100,z5,Soporte_final\WObj:=ADwob;
        MoveL Target_480,v100,z5,Soporte_final\WObj:=ADwob;
        MoveL Target_490,v100,z5,Soporte_final\WObj:=ADwob;
        MoveL Target_460,v100,z5,Soporte_final\WObj:=ADwob;
        MoveL Target_450,v100,z5,Soporte_final\WObj:=ADwob;
        MoveL Target_500,v100,z5,Soporte_final\WObj:=ADwob;
        MoveL Target_510,v100,z5,Soporte_final\WObj:=ADwob;
        MoveL Target_520,v100,z5,Soporte_final\WObj:=ADwob;
        MoveL Target_530,v100,z5,Soporte_final\WObj:=ADwob;
        MoveL Target_540,v100,z5,Soporte_final\WObj:=ADwob;
        MoveL Target_550,v100,z5,Soporte_final\WObj:=ADwob;
        MoveL Target_560,v100,z5,Soporte_final\WObj:=ADwob;
        MoveL Target_570,v100,z5,Soporte_final\WObj:=ADwob;
        MoveL Target_580,v100,z5,Soporte_final\WObj:=ADwob;
        MoveL Target_590,v100,z5,Soporte_final\WObj:=ADwob;
        MoveL Target_500,v100,z5,Soporte_final\WObj:=ADwob;
        MoveL Target_600,v100,z5,Soporte_final\WObj:=ADwob;
        MoveL Target_610,v100,z5,Soporte_final\WObj:=ADwob; !baja en z letra 2 a
        MoveL Target_620,v100,z5,Soporte_final\WObj:=ADwob;
        MoveL Target_630,v100,z5,Soporte_final\WObj:=ADwob;
        MoveL Target_640,v100,z5,Soporte_final\WObj:=ADwob;
        MoveL Target_650,v100,z5,Soporte_final\WObj:=ADwob;
        MoveL Target_660,v100,z5,Soporte_final\WObj:=ADwob;
        MoveL Target_670,v100,z5,Soporte_final\WObj:=ADwob;
        MoveL Target_680,v100,z5,Soporte_final\WObj:=ADwob;
        MoveL Target_690,v100,z5,Soporte_final\WObj:=ADwob;
        MoveL Target_700,v100,z5,Soporte_final\WObj:=ADwob;
        MoveL Target_710,v100,z5,Soporte_final\WObj:=ADwob;
        MoveL Target_720,v100,z5,Soporte_final\WObj:=ADwob;
        MoveL Target_730,v100,z5,Soporte_final\WObj:=ADwob;
        MoveL Target_740,v100,z5,Soporte_final\WObj:=ADwob;
        MoveL Target_750,v100,z5,Soporte_final\WObj:=ADwob;
        MoveL Target_760,v100,z5,Soporte_final\WObj:=ADwob;
        MoveL Target_770,v100,z5,Soporte_final\WObj:=ADwob;
        MoveL Target_780,v100,z5,Soporte_final\WObj:=ADwob;
        MoveL Target_790,v100,z5,Soporte_final\WObj:=ADwob;
        MoveL Target_800,v100,z5,Soporte_final\WObj:=ADwob;
        MoveL Target_810,v100,z5,Soporte_final\WObj:=ADwob;
        MoveL Target_820,v100,z5,Soporte_final\WObj:=ADwob;
        MoveL Target_830,v100,z5,Soporte_final\WObj:=ADwob;
        MoveL Target_840,v100,z5,Soporte_final\WObj:=ADwob;
        MoveL Target_850,v100,z5,Soporte_final\WObj:=ADwob;
        MoveL Target_860,v100,z5,Soporte_final\WObj:=ADwob;
        MoveL Target_870,v100,z5,Soporte_final\WObj:=ADwob;
        MoveL Target_880,v100,z5,Soporte_final\WObj:=ADwob;
        MoveL Target_890,v100,z5,Soporte_final\WObj:=ADwob;
        MoveL Target_900,v100,z5,Soporte_final\WObj:=ADwob;
        MoveL Target_610,v100,z5,Soporte_final\WObj:=ADwob; !une las cosas en a
        MoveL Target_600,v100,z5,Soporte_final\WObj:=ADwob;
        MoveL Target_910,v100,z5,Soporte_final\WObj:=ADwob;
        MoveL Target_920,v100,z5,Soporte_final\WObj:=ADwob;
        MoveL Target_930,v100,z5,Soporte_final\WObj:=ADwob;
        MoveL Target_940,v100,z5,Soporte_final\WObj:=ADwob;
        MoveL Target_950,v100,z5,Soporte_final\WObj:=ADwob;
        MoveL Target_960,v100,z5,Soporte_final\WObj:=ADwob;
        MoveL Target_970,v100,z5,Soporte_final\WObj:=ADwob;
        MoveL Target_980,v100,z5,Soporte_final\WObj:=ADwob;
        MoveL Target_990,v100,z5,Soporte_final\WObj:=ADwob;
        MoveL Target_1000,v100,z5,Soporte_final\WObj:=ADwob;
        MoveL Target_1010,v100,z5,Soporte_final\WObj:=ADwob;
        MoveL Target_1020,v100,z5,Soporte_final\WObj:=ADwob;
        MoveL Target_1030,v100,z5,Soporte_final\WObj:=ADwob;
        MoveL Target_1040,v100,z5,Soporte_final\WObj:=ADwob;
        MoveL Target_1050,v100,z5,Soporte_final\WObj:=ADwob;
        MoveL Target_1060,v100,z5,Soporte_final\WObj:=ADwob;
        MoveL Target_1070,v100,z5,Soporte_final\WObj:=ADwob;
        MoveL Target_1080,v100,z5,Soporte_final\WObj:=ADwob;
        MoveL Target_1090,v100,z5,Soporte_final\WObj:=ADwob;
        MoveL Target_1100,v100,z5,Soporte_final\WObj:=ADwob;
        MoveL Target_920,v100,z5,Soporte_final\WObj:=ADwob;
        MoveL Target_910,v100,z5,Soporte_final\WObj:=ADwob;
        MoveL Target_1110,v100,z5,Soporte_final\WObj:=ADwob;
        MoveL Target_1120,v100,z5,Soporte_final\WObj:=ADwob;
        MoveL Target_1130,v100,z5,Soporte_final\WObj:=ADwob;
        MoveL Target_1140,v100,z5,Soporte_final\WObj:=ADwob;
        MoveL Target_1150,v100,z5,Soporte_final\WObj:=ADwob;
        MoveL Target_1160,v100,z5,Soporte_final\WObj:=ADwob;
        MoveL Target_1170,v100,z5,Soporte_final\WObj:=ADwob;
        MoveL Target_1180,v100,z5,Soporte_final\WObj:=ADwob;
        MoveL Target_1190,v100,z5,Soporte_final\WObj:=ADwob;
        MoveL Target_1200,v100,z5,Soporte_final\WObj:=ADwob;
        MoveL Target_1210,v100,z5,Soporte_final\WObj:=ADwob;
        MoveL Target_1220,v100,z5,Soporte_final\WObj:=ADwob;
        MoveL Target_1230,v100,z5,Soporte_final\WObj:=ADwob;
        MoveL Target_1240,v100,z5,Soporte_final\WObj:=ADwob;
        MoveL Target_1250,v100,z5,Soporte_final\WObj:=ADwob;
        MoveL Target_1260,v100,z5,Soporte_final\WObj:=ADwob;
        MoveL Target_1270,v100,z5,Soporte_final\WObj:=ADwob;
        MoveL Target_1280,v100,z5,Soporte_final\WObj:=ADwob;
        MoveL Target_1290,v100,z5,Soporte_final\WObj:=ADwob;
        MoveL Target_1300,v100,z5,Soporte_final\WObj:=ADwob;
        MoveL Target_1310,v100,z5,Soporte_final\WObj:=ADwob;
        MoveL Target_1320,v100,z5,Soporte_final\WObj:=ADwob;
        MoveL Target_1330,v100,z5,Soporte_final\WObj:=ADwob;
        MoveL Target_1340,v100,z5,Soporte_final\WObj:=ADwob;
        MoveL Target_1350,v100,z5,Soporte_final\WObj:=ADwob;
        MoveL Target_1360,v100,z5,Soporte_final\WObj:=ADwob;
        MoveL Target_1120,v100,z5,Soporte_final\WObj:=ADwob;
        MoveL Target_1110,v100,z5,Soporte_final\WObj:=ADwob;
        MoveL Target_1370,v100,z5,Soporte_final\WObj:=ADwob;
        MoveL Target_1380,v100,z5,Soporte_final\WObj:=ADwob;
        MoveL Target_1390,v100,z5,Soporte_final\WObj:=ADwob;
        MoveL Target_1400,v100,z5,Soporte_final\WObj:=ADwob;
        MoveL Target_1410,v100,z5,Soporte_final\WObj:=ADwob;
        MoveL Target_1420,v100,z5,Soporte_final\WObj:=ADwob;
        MoveL Target_1430,v100,z5,Soporte_final\WObj:=ADwob;
        MoveL Target_1440,v100,z5,Soporte_final\WObj:=ADwob;
        MoveL Target_1450,v100,z5,Soporte_final\WObj:=ADwob;
        MoveL Target_1460,v100,z5,Soporte_final\WObj:=ADwob;
        MoveL Target_1470,v100,z5,Soporte_final\WObj:=ADwob;
        MoveL Target_1480,v100,z5,Soporte_final\WObj:=ADwob;
        MoveL Target_1490,v100,z5,Soporte_final\WObj:=ADwob;
        MoveL Target_1500,v100,z5,Soporte_final\WObj:=ADwob;
        MoveL Target_1510,v100,z5,Soporte_final\WObj:=ADwob;
        MoveL Target_1520,v100,z5,Soporte_final\WObj:=ADwob;
        MoveL Target_1530,v100,z5,Soporte_final\WObj:=ADwob;
        MoveL Target_1540,v100,z5,Soporte_final\WObj:=ADwob;
        MoveL Target_1550,v100,z5,Soporte_final\WObj:=ADwob;
        MoveL Target_1560,v100,z5,Soporte_final\WObj:=ADwob;
        MoveL Target_1570,v100,z5,Soporte_final\WObj:=ADwob;
        MoveL Target_1580,v100,z5,Soporte_final\WObj:=ADwob;
        MoveL Target_1590,v100,z5,Soporte_final\WObj:=ADwob;
        MoveL Target_1600,v100,z5,Soporte_final\WObj:=ADwob;
        MoveL Target_1610,v100,z5,Soporte_final\WObj:=ADwob;
        MoveL Target_1620,v100,z5,Soporte_final\WObj:=ADwob;
        MoveL Target_1630,v100,z5,Soporte_final\WObj:=ADwob;
        MoveL Target_1640,v100,z5,Soporte_final\WObj:=ADwob;
        MoveL Target_1650,v100,z5,Soporte_final\WObj:=ADwob;
        MoveL Target_1660,v100,z5,Soporte_final\WObj:=ADwob;
        MoveL Target_1670,v100,z5,Soporte_final\WObj:=ADwob;
        MoveL Target_1680,v100,z5,Soporte_final\WObj:=ADwob;
        MoveL Target_1690,v100,z5,Soporte_final\WObj:=ADwob;
        MoveL Target_1700,v100,z5,Soporte_final\WObj:=ADwob;
        MoveL Target_1710,v100,z5,Soporte_final\WObj:=ADwob;
        MoveL Target_1720,v100,z5,Soporte_final\WObj:=ADwob;
        MoveL Target_1730,v100,z5,Soporte_final\WObj:=ADwob;
        MoveL Target_1740,v100,z5,Soporte_final\WObj:=ADwob;
        MoveL Target_1750,v100,z5,Soporte_final\WObj:=ADwob;
        MoveL Target_1760,v100,z5,Soporte_final\WObj:=ADwob;
        MoveL Target_1770,v100,z5,Soporte_final\WObj:=ADwob;
        MoveL Target_1780,v100,z5,Soporte_final\WObj:=ADwob;
        MoveL Target_1790,v100,z5,Soporte_final\WObj:=ADwob;
        MoveL Target_1800,v100,z5,Soporte_final\WObj:=ADwob;
        MoveL Target_1810,v100,z5,Soporte_final\WObj:=ADwob;
        MoveL Target_1820,v100,z5,Soporte_final\WObj:=ADwob;
        MoveL Target_1830,v100,z5,Soporte_final\WObj:=ADwob;
        MoveL Target_1840,v100,z5,Soporte_final\WObj:=ADwob;
        MoveL Target_1850,v100,z5,Soporte_final\WObj:=ADwob;
        MoveL Target_1860,v100,z5,Soporte_final\WObj:=ADwob;
        MoveL Target_1870,v100,z5,Soporte_final\WObj:=ADwob;
        MoveL Target_1880,v100,z5,Soporte_final\WObj:=ADwob;
        MoveL Target_1890,v100,z5,Soporte_final\WObj:=ADwob;
        MoveL Target_1900,v100,z5,Soporte_final\WObj:=ADwob;
        MoveL Target_1910,v100,z5,Soporte_final\WObj:=ADwob;
        MoveL Target_1920,v100,z5,Soporte_final\WObj:=ADwob;
        MoveL Target_1930,v100,z5,Soporte_final\WObj:=ADwob;
        MoveL Target_1940,v100,z5,Soporte_final\WObj:=ADwob;
        MoveL Target_1950,v100,z5,Soporte_final\WObj:=ADwob;
        MoveL Target_1960,v100,z5,Soporte_final\WObj:=ADwob;
        MoveL Target_1970,v100,z5,Soporte_final\WObj:=ADwob;
        MoveL Target_1980,v100,z5,Soporte_final\WObj:=ADwob;
        MoveL Target_1990,v100,z5,Soporte_final\WObj:=ADwob;
        MoveL Target_2000,v100,z5,Soporte_final\WObj:=ADwob;
        MoveL Target_2010,v100,z5,Soporte_final\WObj:=ADwob;
        MoveL Target_2020,v100,z5,Soporte_final\WObj:=ADwob;
        MoveL Target_2030,v100,z5,Soporte_final\WObj:=ADwob;
        MoveL Target_2040,v100,z5,Soporte_final\WObj:=ADwob;
        MoveL Target_2050,v100,z5,Soporte_final\WObj:=ADwob;
        MoveL Target_2060,v100,z5,Soporte_final\WObj:=ADwob;
        MoveL Target_2070,v100,z5,Soporte_final\WObj:=ADwob;
        MoveL Target_2080,v100,z5,Soporte_final\WObj:=ADwob;
        MoveL Target_2090,v100,z5,Soporte_final\WObj:=ADwob;
        MoveL Target_2100,v100,z5,Soporte_final\WObj:=ADwob;
        MoveL Target_2110,v100,z5,Soporte_final\WObj:=ADwob;
        MoveL Target_2120,v100,z5,Soporte_final\WObj:=ADwob;
        MoveL Target_2130,v100,z5,Soporte_final\WObj:=ADwob;
        MoveL Target_2140,v100,z5,Soporte_final\WObj:=ADwob;
        MoveL Target_2150,v100,z5,Soporte_final\WObj:=ADwob;
        MoveL Target_2160,v100,z5,Soporte_final\WObj:=ADwob;
        MoveL Target_2170,v100,z5,Soporte_final\WObj:=ADwob;
        MoveL Target_2180,v100,z5,Soporte_final\WObj:=ADwob;
        MoveL Target_2190,v100,z5,Soporte_final\WObj:=ADwob;
        MoveL Target_2200,v100,z5,Soporte_final\WObj:=ADwob;
        MoveL Target_2210,v100,z5,Soporte_final\WObj:=ADwob;
        MoveL Target_2220,v100,z5,Soporte_final\WObj:=ADwob;
        MoveL Target_2230,v100,z5,Soporte_final\WObj:=ADwob;
        MoveL Target_2240,v100,z5,Soporte_final\WObj:=ADwob;
        MoveL Target_1380,v100,z5,Soporte_final\WObj:=ADwob; !une letra a ultima
        MoveL Target_1370,v100,z5,Soporte_final\WObj:=ADwob; !sube en z
        MoveL Target_2250,v100,z5,Soporte_final\WObj:=ADwob; !circulos de las cosas
        MoveL Target_2260,v100,z5,Soporte_final\WObj:=ADwob;  !baja en z
        MoveL Target_2270,v100,z5,Soporte_final\WObj:=ADwob;
        MoveL Target_2280,v100,z5,Soporte_final\WObj:=ADwob;
        MoveL Target_2290,v100,z5,Soporte_final\WObj:=ADwob;
        MoveL Target_2300,v100,z5,Soporte_final\WObj:=ADwob;
        MoveL Target_2310,v100,z5,Soporte_final\WObj:=ADwob;
        MoveL Target_2320,v100,z5,Soporte_final\WObj:=ADwob;
        MoveL Target_2340,v100,z5,Soporte_final\WObj:=ADwob;
        MoveL Target_2350,v100,z5,Soporte_final\WObj:=ADwob;
        MoveL Target_2360,v100,z5,Soporte_final\WObj:=ADwob;
        MoveL Target_2370,v100,z5,Soporte_final\WObj:=ADwob;
        MoveL Target_2380,v100,z5,Soporte_final\WObj:=ADwob;
        MoveL Target_2390,v100,z5,Soporte_final\WObj:=ADwob;
        MoveL Target_2400,v100,z5,Soporte_final\WObj:=ADwob;
        MoveL Target_2410,v100,z5,Soporte_final\WObj:=ADwob;
        MoveL Target_2420,v100,z5,Soporte_final\WObj:=ADwob;
        MoveL Target_2430,v100,z5,Soporte_final\WObj:=ADwob;
        MoveL Target_2440,v100,z5,Soporte_final\WObj:=ADwob;
        MoveL Target_2450,v100,z5,Soporte_final\WObj:=ADwob;
        MoveL Target_2460,v100,z5,Soporte_final\WObj:=ADwob;
        MoveL Target_2470,v100,z5,Soporte_final\WObj:=ADwob;
        MoveL Target_2260,v100,z5,Soporte_final\WObj:=ADwob; !cierra circulo de a
        MoveL Target_2250,v100,z5,Soporte_final\WObj:=ADwob; !sube en z
        MoveL Target_2330,v100,z5,Soporte_final\WObj:=ADwob; !llega arriba en d
        MoveL Target_2500,v100,z5,Soporte_final\WObj:=ADwob;
        MoveL Target_2510,v100,z5,Soporte_final\WObj:=ADwob;
        MoveL Target_2520,v100,z5,Soporte_final\WObj:=ADwob;
        MoveL Target_2530,v100,z5,Soporte_final\WObj:=ADwob;
        MoveL Target_2540,v100,z5,Soporte_final\WObj:=ADwob;
        MoveL Target_2550,v100,z5,Soporte_final\WObj:=ADwob;
        MoveL Target_2560,v100,z5,Soporte_final\WObj:=ADwob;
        MoveL Target_2570,v100,z5,Soporte_final\WObj:=ADwob;
        MoveL Target_2580,v100,z5,Soporte_final\WObj:=ADwob;
        MoveL Target_2590,v100,z5,Soporte_final\WObj:=ADwob;
        MoveL Target_2600,v100,z5,Soporte_final\WObj:=ADwob;
        MoveL Target_2610,v100,z5,Soporte_final\WObj:=ADwob;
        MoveL Target_2620,v100,z5,Soporte_final\WObj:=ADwob;
        MoveL Target_2630,v100,z5,Soporte_final\WObj:=ADwob;
        MoveL Target_2640,v100,z5,Soporte_final\WObj:=ADwob;
        MoveL Target_2650,v100,z5,Soporte_final\WObj:=ADwob;
        MoveL Target_2660,v100,z5,Soporte_final\WObj:=ADwob;
        MoveL Target_2670,v100,z5,Soporte_final\WObj:=ADwob;
        MoveL Target_2690,v100,z5,Soporte_final\WObj:=ADwob;
        MoveL Target_2700,v100,z5,Soporte_final\WObj:=ADwob;
        MoveL Target_2710,v100,z5,Soporte_final\WObj:=ADwob;
        MoveL Target_2720,v100,z5,Soporte_final\WObj:=ADwob;
        MoveL Target_2730,v100,z5,Soporte_final\WObj:=ADwob;
        MoveL Target_2740,v100,z5,Soporte_final\WObj:=ADwob;
        MoveL Target_2750,v100,z5,Soporte_final\WObj:=ADwob;
        MoveL Target_2500,v100,z5,Soporte_final\WObj:=ADwob;
        MoveL Target_2330,v100,z5,Soporte_final\WObj:=ADwob;
        MoveL Target_2760,v100,z5,Soporte_final\WObj:=ADwob;
        MoveL Target_2770,v100,z5,Soporte_final\WObj:=ADwob;
        MoveL Target_2780,v100,z5,Soporte_final\WObj:=ADwob;
        MoveL Target_2790,v100,z5,Soporte_final\WObj:=ADwob;
        MoveL Target_2800,v100,z5,Soporte_final\WObj:=ADwob;
        MoveL Target_2810,v100,z5,Soporte_final\WObj:=ADwob;
        MoveL Target_2820,v100,z5,Soporte_final\WObj:=ADwob;
        MoveL Target_2830,v100,z5,Soporte_final\WObj:=ADwob;
        MoveL Target_2840,v100,z5,Soporte_final\WObj:=ADwob;
        MoveL Target_2850,v100,z5,Soporte_final\WObj:=ADwob;
        MoveL Target_2860,v100,z5,Soporte_final\WObj:=ADwob;
        MoveL Target_2870,v100,z5,Soporte_final\WObj:=ADwob;
        MoveL Target_2880,v100,z5,Soporte_final\WObj:=ADwob;
        MoveL Target_2890,v100,z5,Soporte_final\WObj:=ADwob;
        MoveL Target_2900,v100,z5,Soporte_final\WObj:=ADwob;
        MoveL Target_2910,v100,z5,Soporte_final\WObj:=ADwob;
        MoveL Target_2770,v100,z5,Soporte_final\WObj:=ADwob;
        MoveL Target_2760,v100,z5,Soporte_final\WObj:=ADwob; ! queda arriba final.
        MoveJ Target_minihome,v100,z5,Soporte_final\WObj:=ADwob;
    ENDPROC
    PROC Path_20()
        MoveJ Target_minihome,v100,z5,Soporte_final\WObj:=ADwob;
        MoveL Target_2920_up,v100,z5,Soporte_final\WObj:=ADwob;
        MoveL Target_2920,v100,z5,Soporte_final\WObj:=ADwob;
        MoveL Target_2930,v100,z5,Soporte_final\WObj:=ADwob;
        MoveC Target_2940,Target_2950,v100,z5,Soporte_final\WObj:=ADwob;
        MoveL Target_2960,v100,z5,Soporte_final\WObj:=ADwob;
                MoveL Target_2920,v100,z5,Soporte_final\WObj:=ADwob;
        MoveL Target_2970_up,v100,z5,Soporte_final\WObj:=ADwob;
        MoveL Target_2970,v100,z5,Soporte_final\WObj:=ADwob;
        MoveL Target_2980,v100,z5,Soporte_final\WObj:=ADwob;
        MoveC Target_2990,Target_3000,v100,z5,Soporte_final\WObj:=ADwob;
        MoveL Target_3010,v100,z5,Soporte_final\WObj:=ADwob;
                MoveL Target_2970,v100,z5,Soporte_final\WObj:=ADwob;
        MoveL Target_3030_2,v100,z5,Soporte_final\WObj:=ADwob;
        MoveL Target_3030,v100,z5,Soporte_final\WObj:=ADwob;
        MoveL Target_3040,v100,z5,Soporte_final\WObj:=ADwob;
        MoveL Target_3050,v100,z5,Soporte_final\WObj:=ADwob;
        MoveL Target_3060,v100,z5,Soporte_final\WObj:=ADwob;
        MoveL Target_3070,v100,z5,Soporte_final\WObj:=ADwob;
        MoveL Target_3080,v100,z5,Soporte_final\WObj:=ADwob;
        MoveL Target_3090,v100,z5,Soporte_final\WObj:=ADwob;
        MoveL Target_3100,v100,z5,Soporte_final\WObj:=ADwob;
        MoveL Target_3110,v100,z5,Soporte_final\WObj:=ADwob;
        MoveL Target_3120,v100,z5,Soporte_final\WObj:=ADwob;
        MoveL Target_3130,v100,z5,Soporte_final\WObj:=ADwob;
        MoveL Target_3140,v100,z5,Soporte_final\WObj:=ADwob;
        MoveL Target_3150,v100,z5,Soporte_final\WObj:=ADwob;
        MoveL Target_3160,v100,z5,Soporte_final\WObj:=ADwob;
        MoveL Target_3170,v100,z5,Soporte_final\WObj:=ADwob;
        MoveL Target_3180,v100,z5,Soporte_final\WObj:=ADwob;
        MoveL Target_3190,v100,z5,Soporte_final\WObj:=ADwob;
        MoveL Target_3200,v100,z5,Soporte_final\WObj:=ADwob;
        MoveL Target_3210,v100,z5,Soporte_final\WObj:=ADwob;
        MoveL Target_3220,v100,z5,Soporte_final\WObj:=ADwob;
        MoveL Target_3230,v100,z5,Soporte_final\WObj:=ADwob;
        MoveL Target_3240,v100,z5,Soporte_final\WObj:=ADwob;
        MoveL Target_3250,v100,z5,Soporte_final\WObj:=ADwob;
        MoveL Target_3030,v100,z5,Soporte_final\WObj:=ADwob;
        MoveL Target_3260_2,v100,z5,Soporte_final\WObj:=ADwob;
        MoveL Target_3260,v100,z5,Soporte_final\WObj:=ADwob;
        MoveL Target_3270,v100,z5,Soporte_final\WObj:=ADwob;
        MoveL Target_3280,v100,z5,Soporte_final\WObj:=ADwob;
        MoveL Target_3290,v100,z5,Soporte_final\WObj:=ADwob;
        MoveL Target_3300,v100,z5,Soporte_final\WObj:=ADwob;
        MoveL Target_3310,v100,z5,Soporte_final\WObj:=ADwob;
        MoveL Target_3320,v100,z5,Soporte_final\WObj:=ADwob;
        MoveL Target_3330,v100,z5,Soporte_final\WObj:=ADwob;
        MoveL Target_3340,v100,z5,Soporte_final\WObj:=ADwob;
        MoveL Target_3260,v100,z5,Soporte_final\WObj:=ADwob;
        MoveL Target_3350_2,v100,z5,Soporte_final\WObj:=ADwob;
        MoveL Target_3350,v100,z5,Soporte_final\WObj:=ADwob;
        MoveL Target_3360,v100,z5,Soporte_final\WObj:=ADwob;
        MoveL Target_3370,v100,z5,Soporte_final\WObj:=ADwob;
        MoveL Target_3380,v100,z5,Soporte_final\WObj:=ADwob;
        MoveL Target_3390,v100,z5,Soporte_final\WObj:=ADwob;
        MoveL Target_3400,v100,z5,Soporte_final\WObj:=ADwob;
        MoveL Target_3410,v100,z5,Soporte_final\WObj:=ADwob;
        MoveL Target_3350,v100,z5,Soporte_final\WObj:=ADwob;
        MoveL Target_3420_2,v100,z5,Soporte_final\WObj:=ADwob;
        MoveL Target_3420,v100,z5,Soporte_final\WObj:=ADwob;
        MoveL Target_3430,v100,z5,Soporte_final\WObj:=ADwob;
        MoveL Target_3440,v100,z5,Soporte_final\WObj:=ADwob;
        MoveL Target_3450,v100,z5,Soporte_final\WObj:=ADwob;
        MoveL Target_3420,v100,z5,Soporte_final\WObj:=ADwob;
        MoveL Target_3460_2,v100,z5,Soporte_final\WObj:=ADwob;
        MoveL Target_3460,v100,z5,Soporte_final\WObj:=ADwob;
        MoveL Target_3470,v100,z5,Soporte_final\WObj:=ADwob;
        MoveL Target_3480,v100,z5,Soporte_final\WObj:=ADwob;
        MoveL Target_3490,v100,z5,Soporte_final\WObj:=ADwob;
        MoveL Target_3500,v100,z5,Soporte_final\WObj:=ADwob;
        MoveL Target_3510,v100,z5,Soporte_final\WObj:=ADwob;
                MoveL Target_3460,v100,z5,Soporte_final\WObj:=ADwob;
                MoveL Target_3520_2,v100,z5,Soporte_final\WObj:=ADwob;
                MoveL Target_3520,v100,z5,Soporte_final\WObj:=ADwob;
        MoveL Target_3530,v100,z5,Soporte_final\WObj:=ADwob;
        MoveL Target_3540,v100,z5,Soporte_final\WObj:=ADwob;
        MoveL Target_3550,v100,z5,Soporte_final\WObj:=ADwob;
        MoveL Target_3560,v100,z5,Soporte_final\WObj:=ADwob;
        MoveL Target_3570,v100,z5,Soporte_final\WObj:=ADwob;
        MoveL Target_3580,v100,z5,Soporte_final\WObj:=ADwob;
                MoveL Target_3590,v100,z5,Soporte_final\WObj:=ADwob;
                MoveL Target_3600,v100,z5,Soporte_final\WObj:=ADwob;
        MoveL Target_3610,v100,z5,Soporte_final\WObj:=ADwob;
        MoveL Target_3620,v100,z5,Soporte_final\WObj:=ADwob;
        MoveL Target_3630,v100,z5,Soporte_final\WObj:=ADwob;
        MoveL Target_3640,v100,z5,Soporte_final\WObj:=ADwob;
        MoveL Target_3650,v100,z5,Soporte_final\WObj:=ADwob;
        MoveL Target_3660,v100,z5,Soporte_final\WObj:=ADwob;
        MoveL Target_3520,v100,z5,Soporte_final\WObj:=ADwob;
                MoveL Target_3670_2,v100,z5,Soporte_final\WObj:=ADwob;
                MoveL Target_3670,v100,z5,Soporte_final\WObj:=ADwob;
                MoveL Target_3680,v100,z5,Soporte_final\WObj:=ADwob;
        MoveL Target_3690,v100,z5,Soporte_final\WObj:=ADwob;
        MoveL Target_3700,v100,z5,Soporte_final\WObj:=ADwob;
        MoveL Target_3710,v100,z5,Soporte_final\WObj:=ADwob;
        MoveL Target_3720,v100,z5,Soporte_final\WObj:=ADwob;
        MoveL Target_3730,v100,z5,Soporte_final\WObj:=ADwob;
        MoveL Target_3740,v100,z5,Soporte_final\WObj:=ADwob;
        MoveL Target_3670,v100,z5,Soporte_final\WObj:=ADwob;
        MoveJ Target_minihome,v100,z5,Soporte_final\WObj:=ADwob;
    ENDPROC
    PROC Path_30()
                MoveL Target_3750_2,v100,z5,Soporte_final\WObj:=ADwob;
        MoveL Target_3750,v100,z5,Soporte_final\WObj:=ADwob;
        MoveL Target_3760,v100,z5,Soporte_final\WObj:=ADwob;
        MoveL Target_3770,v100,z5,Soporte_final\WObj:=ADwob;
        MoveL Target_3780,v100,z5,Soporte_final\WObj:=ADwob;
        MoveL Target_3790,v100,z5,Soporte_final\WObj:=ADwob;
        MoveL Target_3800,v100,z5,Soporte_final\WObj:=ADwob;
        MoveL Target_3810,v100,z5,Soporte_final\WObj:=ADwob;
        MoveL Target_3820,v100,z5,Soporte_final\WObj:=ADwob;
        MoveL Target_3830,v100,z5,Soporte_final\WObj:=ADwob;
        MoveL Target_3840,v100,z5,Soporte_final\WObj:=ADwob;
        MoveL Target_3850,v100,z5,Soporte_final\WObj:=ADwob;
        MoveL Target_3860,v100,z5,Soporte_final\WObj:=ADwob;
        MoveL Target_3870,v100,z5,Soporte_final\WObj:=ADwob;
        MoveL Target_3880,v100,z5,Soporte_final\WObj:=ADwob;
        MoveL Target_3890,v100,z5,Soporte_final\WObj:=ADwob;
        MoveL Target_3900,v100,z5,Soporte_final\WObj:=ADwob;
                MoveL Target_3750,v100,z5,Soporte_final\WObj:=ADwob;
                MoveL Target_3910_2,v100,z5,Soporte_final\WObj:=ADwob;
        MoveL Target_3910,v100,z5,Soporte_final\WObj:=ADwob;
        MoveL Target_3920,v100,z5,Soporte_final\WObj:=ADwob;
        MoveL Target_3930,v100,z5,Soporte_final\WObj:=ADwob;
        MoveL Target_3940,v100,z5,Soporte_final\WObj:=ADwob;
        MoveL Target_3950,v100,z5,Soporte_final\WObj:=ADwob;
        MoveL Target_3960,v100,z5,Soporte_final\WObj:=ADwob;
                MoveL Target_3910,v100,z5,Soporte_final\WObj:=ADwob;
                MoveL Target_3970_2,v100,z5,Soporte_final\WObj:=ADwob;
        MoveL Target_3970,v100,z5,Soporte_final\WObj:=ADwob;
        MoveL Target_3980,v100,z5,Soporte_final\WObj:=ADwob;
        MoveL Target_3990,v100,z5,Soporte_final\WObj:=ADwob;
        MoveL Target_4000,v100,z5,Soporte_final\WObj:=ADwob;
                MoveL Target_3970,v100,z5,Soporte_final\WObj:=ADwob;
                MoveL Target_4010_2,v100,z5,Soporte_final\WObj:=ADwob;
        MoveL Target_4010,v100,z5,Soporte_final\WObj:=ADwob;
        MoveL Target_4020,v100,z5,Soporte_final\WObj:=ADwob;
        MoveL Target_4030,v100,z5,Soporte_final\WObj:=ADwob;
        MoveL Target_4040,v100,z5,Soporte_final\WObj:=ADwob;
        MoveL Target_4050,v100,z5,Soporte_final\WObj:=ADwob;
        MoveL Target_4060,v100,z5,Soporte_final\WObj:=ADwob;
        MoveL Target_4070,v100,z5,Soporte_final\WObj:=ADwob;
        MoveL Target_4080,v100,z5,Soporte_final\WObj:=ADwob;
        MoveL Target_4090,v100,z5,Soporte_final\WObj:=ADwob;
        MoveL Target_4100,v100,z5,Soporte_final\WObj:=ADwob;
        MoveL Target_4110,v100,z5,Soporte_final\WObj:=ADwob;
        MoveL Target_4120,v100,z5,Soporte_final\WObj:=ADwob;
        MoveL Target_4130,v100,z5,Soporte_final\WObj:=ADwob;
        MoveL Target_4010,v100,z5,Soporte_final\WObj:=ADwob;
        MoveL Target_minihome,v100,z5,Soporte_final\WObj:=ADwob;
    ENDPROC


    PROC Path_40()
        MoveJ Target_minihome_2,v100,z5,Soporte_final\WObj:=ADWob_2;
        MoveJ Target_200_2,v100,z5,Soporte_final\WObj:=ADWob_2;
        MoveL Target_210_2,v100,z5,Soporte_final\WObj:=ADWob_2;
        MoveL Target_220_2,v100,z5,Soporte_final\WObj:=ADWob_2;
        MoveL Target_230_2,v100,z5,Soporte_final\WObj:=ADWob_2;
        MoveL Target_240_2,v100,z5,Soporte_final\WObj:=ADWob_2;
        MoveL Target_250_2,v100,z5,Soporte_final\WObj:=ADWob_2;
        MoveL Target_260_2,v100,z5,Soporte_final\WObj:=ADWob_2;
        MoveL Target_270_2,v100,z5,Soporte_final\WObj:=ADWob_2;
        MoveL Target_280_2,v100,z5,Soporte_final\WObj:=ADWob_2;
        MoveL Target_210_2,v100,z5,Soporte_final\WObj:=ADWob_2;
        MoveL Target_200_2,v100,z5,Soporte_final\WObj:=ADWob_2;
        MoveL Target_290_2,v100,z5,Soporte_final\WObj:=ADWob_2;
        MoveL Target_300_2,v100,z5,Soporte_final\WObj:=ADWob_2;
        MoveL Target_310_2,v100,z5,Soporte_final\WObj:=ADWob_2;
        MoveL Target_320_2,v100,z5,Soporte_final\WObj:=ADWob_2;
        MoveL Target_300_2,v100,z5,Soporte_final\WObj:=ADWob_2;
        MoveL Target_290_2,v100,z5,Soporte_final\WObj:=ADWob_2;
        MoveL Target_330_2,v100,z5,Soporte_final\WObj:=ADWob_2;
        MoveL Target_340_2,v100,z5,Soporte_final\WObj:=ADWob_2;
        MoveL Target_350_2,v100,z5,Soporte_final\WObj:=ADWob_2;
        MoveL Target_360_2,v100,z5,Soporte_final\WObj:=ADWob_2;
        MoveL Target_370_2,v100,z5,Soporte_final\WObj:=ADWob_2;
        MoveL Target_380_2,v100,z5,Soporte_final\WObj:=ADWob_2;
        MoveL Target_390_2,v100,z5,Soporte_final\WObj:=ADWob_2;
        MoveL Target_400_2,v100,z5,Soporte_final\WObj:=ADWob_2;
        MoveL Target_410_2,v100,z5,Soporte_final\WObj:=ADWob_2;
        MoveL Target_420_2,v100,z5,Soporte_final\WObj:=ADWob_2;
        MoveL Target_430_2,v100,z5,Soporte_final\WObj:=ADWob_2;
        MoveL Target_440_2,v100,z5,Soporte_final\WObj:=ADWob_2;
        MoveL Target_340_2,v100,z5,Soporte_final\WObj:=ADWob_2;
        MoveL Target_330_2,v100,z5,Soporte_final\WObj:=ADWob_2;
        MoveL Target_450_2,v100,z5,Soporte_final\WObj:=ADWob_2;
        MoveL Target_460_2,v100,z5,Soporte_final\WObj:=ADWob_2;
        MoveL Target_470_2,v100,z5,Soporte_final\WObj:=ADWob_2;
        MoveL Target_480_2,v100,z5,Soporte_final\WObj:=ADWob_2;
        MoveL Target_490_2,v100,z5,Soporte_final\WObj:=ADWob_2;
        MoveL Target_460_2,v100,z5,Soporte_final\WObj:=ADWob_2;
        MoveL Target_450_2,v100,z5,Soporte_final\WObj:=ADWob_2;
        MoveL Target_500_2,v100,z5,Soporte_final\WObj:=ADWob_2;
        MoveL Target_510_2,v100,z5,Soporte_final\WObj:=ADWob_2;
        MoveL Target_520_2,v100,z5,Soporte_final\WObj:=ADWob_2;
        MoveL Target_530_2,v100,z5,Soporte_final\WObj:=ADWob_2;
        MoveL Target_540_2,v100,z5,Soporte_final\WObj:=ADWob_2;
        MoveL Target_550_2,v100,z5,Soporte_final\WObj:=ADWob_2;
        MoveL Target_560_2,v100,z5,Soporte_final\WObj:=ADWob_2;
        MoveL Target_570_2,v100,z5,Soporte_final\WObj:=ADWob_2;
        MoveL Target_580_2,v100,z5,Soporte_final\WObj:=ADWob_2;
        MoveL Target_590_2,v100,z5,Soporte_final\WObj:=ADWob_2;
        MoveL Target_500_2,v100,z5,Soporte_final\WObj:=ADWob_2;
        MoveL Target_600_2,v100,z5,Soporte_final\WObj:=ADWob_2;
        MoveL Target_610_2,v100,z5,Soporte_final\WObj:=ADWob_2; !baja en z letra 2 a
        MoveL Target_620_2,v100,z5,Soporte_final\WObj:=ADWob_2;
        MoveL Target_630_2,v100,z5,Soporte_final\WObj:=ADWob_2;
        MoveL Target_640_2,v100,z5,Soporte_final\WObj:=ADWob_2;
        MoveL Target_650_2,v100,z5,Soporte_final\WObj:=ADWob_2;
        MoveL Target_660_2,v100,z5,Soporte_final\WObj:=ADWob_2;
        MoveL Target_670_2,v100,z5,Soporte_final\WObj:=ADWob_2;
        MoveL Target_680_2,v100,z5,Soporte_final\WObj:=ADWob_2;
        MoveL Target_690_2,v100,z5,Soporte_final\WObj:=ADWob_2;
        MoveL Target_700_2,v100,z5,Soporte_final\WObj:=ADWob_2;
        MoveL Target_710_2,v100,z5,Soporte_final\WObj:=ADWob_2;
        MoveL Target_720_2,v100,z5,Soporte_final\WObj:=ADWob_2;
        MoveL Target_730_2,v100,z5,Soporte_final\WObj:=ADWob_2;
        MoveL Target_740_2,v100,z5,Soporte_final\WObj:=ADWob_2;
        MoveL Target_750_2,v100,z5,Soporte_final\WObj:=ADWob_2;
        MoveL Target_760_2,v100,z5,Soporte_final\WObj:=ADWob_2;
        MoveL Target_770_2,v100,z5,Soporte_final\WObj:=ADWob_2;
        MoveL Target_780_2,v100,z5,Soporte_final\WObj:=ADWob_2;
        MoveL Target_790_2,v100,z5,Soporte_final\WObj:=ADWob_2;
        MoveL Target_800_2,v100,z5,Soporte_final\WObj:=ADWob_2;
        MoveL Target_810_2,v100,z5,Soporte_final\WObj:=ADWob_2;
        MoveL Target_820_2,v100,z5,Soporte_final\WObj:=ADWob_2;
        MoveL Target_830_2,v100,z5,Soporte_final\WObj:=ADWob_2;
        MoveL Target_840_2,v100,z5,Soporte_final\WObj:=ADWob_2;
        MoveL Target_850_2,v100,z5,Soporte_final\WObj:=ADWob_2;
        MoveL Target_860_2,v100,z5,Soporte_final\WObj:=ADWob_2;
        MoveL Target_870_2,v100,z5,Soporte_final\WObj:=ADWob_2;
        MoveL Target_880_2,v100,z5,Soporte_final\WObj:=ADWob_2;
        MoveL Target_890_2,v100,z5,Soporte_final\WObj:=ADWob_2;
        MoveL Target_900_2,v100,z5,Soporte_final\WObj:=ADWob_2;
        MoveL Target_610_2,v100,z5,Soporte_final\WObj:=ADWob_2; !une las cosas en a
        MoveL Target_600_2,v100,z5,Soporte_final\WObj:=ADWob_2;
        MoveL Target_910_2,v100,z5,Soporte_final\WObj:=ADWob_2;
        MoveL Target_920_2,v100,z5,Soporte_final\WObj:=ADWob_2;
        MoveL Target_930_2,v100,z5,Soporte_final\WObj:=ADWob_2;
        MoveL Target_940_2,v100,z5,Soporte_final\WObj:=ADWob_2;
        MoveL Target_950_2,v100,z5,Soporte_final\WObj:=ADWob_2;
        MoveL Target_960_2,v100,z5,Soporte_final\WObj:=ADWob_2;
        MoveL Target_970_2,v100,z5,Soporte_final\WObj:=ADWob_2;
        MoveL Target_980_2,v100,z5,Soporte_final\WObj:=ADWob_2;
        MoveL Target_990_2,v100,z5,Soporte_final\WObj:=ADWob_2;
        MoveL Target_1000_2,v100,z5,Soporte_final\WObj:=ADWob_2;
        MoveL Target_1010_2,v100,z5,Soporte_final\WObj:=ADWob_2;
        MoveL Target_1020_2,v100,z5,Soporte_final\WObj:=ADWob_2;
        MoveL Target_1030_2,v100,z5,Soporte_final\WObj:=ADWob_2;
        MoveL Target_1040_2,v100,z5,Soporte_final\WObj:=ADWob_2;
        MoveL Target_1050_2,v100,z5,Soporte_final\WObj:=ADWob_2;
        MoveL Target_1060_2,v100,z5,Soporte_final\WObj:=ADWob_2;
        MoveL Target_1070_2,v100,z5,Soporte_final\WObj:=ADWob_2;
        MoveL Target_1080_2,v100,z5,Soporte_final\WObj:=ADWob_2;
        MoveL Target_1090_2,v100,z5,Soporte_final\WObj:=ADWob_2;
        MoveL Target_1100_2,v100,z5,Soporte_final\WObj:=ADWob_2;
        MoveL Target_920_2,v100,z5,Soporte_final\WObj:=ADWob_2;
        MoveL Target_910_2,v100,z5,Soporte_final\WObj:=ADWob_2;
        MoveL Target_1110_2,v100,z5,Soporte_final\WObj:=ADWob_2;
        MoveL Target_1120_2,v100,z5,Soporte_final\WObj:=ADWob_2;
        MoveL Target_1130_2,v100,z5,Soporte_final\WObj:=ADWob_2;
        MoveL Target_1140_2,v100,z5,Soporte_final\WObj:=ADWob_2;
        MoveL Target_1150_2,v100,z5,Soporte_final\WObj:=ADWob_2;
        MoveL Target_1160_2,v100,z5,Soporte_final\WObj:=ADWob_2;
        MoveL Target_1170_2,v100,z5,Soporte_final\WObj:=ADWob_2;
        MoveL Target_1180_2,v100,z5,Soporte_final\WObj:=ADWob_2;
        MoveL Target_1190_2,v100,z5,Soporte_final\WObj:=ADWob_2;
        MoveL Target_1200_2,v100,z5,Soporte_final\WObj:=ADWob_2;
        MoveL Target_1210_2,v100,z5,Soporte_final\WObj:=ADWob_2;
        MoveL Target_1220_2,v100,z5,Soporte_final\WObj:=ADWob_2;
        MoveL Target_1230_2,v100,z5,Soporte_final\WObj:=ADWob_2;
        MoveL Target_1240_2,v100,z5,Soporte_final\WObj:=ADWob_2;
        MoveL Target_1250_2,v100,z5,Soporte_final\WObj:=ADWob_2;
        MoveL Target_1260_2,v100,z5,Soporte_final\WObj:=ADWob_2;
        MoveL Target_1270_2,v100,z5,Soporte_final\WObj:=ADWob_2;
        MoveL Target_1280_2,v100,z5,Soporte_final\WObj:=ADWob_2;
        MoveL Target_1290_2,v100,z5,Soporte_final\WObj:=ADWob_2;
        MoveL Target_1300_2,v100,z5,Soporte_final\WObj:=ADWob_2;
        MoveL Target_1310_2,v100,z5,Soporte_final\WObj:=ADWob_2;
        MoveL Target_1320_2,v100,z5,Soporte_final\WObj:=ADWob_2;
        MoveL Target_1330_2,v100,z5,Soporte_final\WObj:=ADWob_2;
        MoveL Target_1340_2,v100,z5,Soporte_final\WObj:=ADWob_2;
        MoveL Target_1350_2,v100,z5,Soporte_final\WObj:=ADWob_2;
        MoveL Target_1360_2,v100,z5,Soporte_final\WObj:=ADWob_2;
        MoveL Target_1120_2,v100,z5,Soporte_final\WObj:=ADWob_2;
        MoveL Target_1110_2,v100,z5,Soporte_final\WObj:=ADWob_2;
        MoveL Target_1370_2,v100,z5,Soporte_final\WObj:=ADWob_2;
        MoveL Target_1380_2,v100,z5,Soporte_final\WObj:=ADWob_2;
        MoveL Target_1390_2,v100,z5,Soporte_final\WObj:=ADWob_2;
        MoveL Target_1400_2,v100,z5,Soporte_final\WObj:=ADWob_2;
        MoveL Target_1410_2,v100,z5,Soporte_final\WObj:=ADWob_2;
        MoveL Target_1420_2,v100,z5,Soporte_final\WObj:=ADWob_2;
        MoveL Target_1430_2,v100,z5,Soporte_final\WObj:=ADWob_2;
        MoveL Target_1440_2,v100,z5,Soporte_final\WObj:=ADWob_2;
        MoveL Target_1450_2,v100,z5,Soporte_final\WObj:=ADWob_2;
        MoveL Target_1460_2,v100,z5,Soporte_final\WObj:=ADWob_2;
        MoveL Target_1470_2,v100,z5,Soporte_final\WObj:=ADWob_2;
        MoveL Target_1480_2,v100,z5,Soporte_final\WObj:=ADWob_2;
        MoveL Target_1490_2,v100,z5,Soporte_final\WObj:=ADWob_2;
        MoveL Target_1500_2,v100,z5,Soporte_final\WObj:=ADWob_2;
        MoveL Target_1510_2,v100,z5,Soporte_final\WObj:=ADWob_2;
        MoveL Target_1520_2,v100,z5,Soporte_final\WObj:=ADWob_2;
        MoveL Target_1530_2,v100,z5,Soporte_final\WObj:=ADWob_2;
        MoveL Target_1540_2,v100,z5,Soporte_final\WObj:=ADWob_2;
        MoveL Target_1550_2,v100,z5,Soporte_final\WObj:=ADWob_2;
        MoveL Target_1560_2,v100,z5,Soporte_final\WObj:=ADWob_2;
        MoveL Target_1570_2,v100,z5,Soporte_final\WObj:=ADWob_2;
        MoveL Target_1580_2,v100,z5,Soporte_final\WObj:=ADWob_2;
        MoveL Target_1590_2,v100,z5,Soporte_final\WObj:=ADWob_2;
        MoveL Target_1600_2,v100,z5,Soporte_final\WObj:=ADWob_2;
        MoveL Target_1610_2,v100,z5,Soporte_final\WObj:=ADWob_2;
        MoveL Target_1620_2,v100,z5,Soporte_final\WObj:=ADWob_2;
        MoveL Target_1630_2,v100,z5,Soporte_final\WObj:=ADWob_2;
        MoveL Target_1640_2,v100,z5,Soporte_final\WObj:=ADWob_2;
        MoveL Target_1650_2,v100,z5,Soporte_final\WObj:=ADWob_2;
        MoveL Target_1660_2,v100,z5,Soporte_final\WObj:=ADWob_2;
        MoveL Target_1670_2,v100,z5,Soporte_final\WObj:=ADWob_2;
        MoveL Target_1680_2,v100,z5,Soporte_final\WObj:=ADWob_2;
        MoveL Target_1690_2,v100,z5,Soporte_final\WObj:=ADWob_2;
        MoveL Target_1700_2,v100,z5,Soporte_final\WObj:=ADWob_2;
        MoveL Target_1710_2,v100,z5,Soporte_final\WObj:=ADWob_2;
        MoveL Target_1720_2,v100,z5,Soporte_final\WObj:=ADWob_2;
        MoveL Target_1730_2,v100,z5,Soporte_final\WObj:=ADWob_2;
        MoveL Target_1740_2,v100,z5,Soporte_final\WObj:=ADWob_2;
        MoveL Target_1750_2,v100,z5,Soporte_final\WObj:=ADWob_2;
        MoveL Target_1760_2,v100,z5,Soporte_final\WObj:=ADWob_2;
        MoveL Target_1770_2,v100,z5,Soporte_final\WObj:=ADWob_2;
        MoveL Target_1780_2,v100,z5,Soporte_final\WObj:=ADWob_2;
        MoveL Target_1790_2,v100,z5,Soporte_final\WObj:=ADWob_2;
        MoveL Target_1800_2,v100,z5,Soporte_final\WObj:=ADWob_2;
        MoveL Target_1810_2,v100,z5,Soporte_final\WObj:=ADWob_2;
        MoveL Target_1820_2,v100,z5,Soporte_final\WObj:=ADWob_2;
        MoveL Target_1830_2,v100,z5,Soporte_final\WObj:=ADWob_2;
        MoveL Target_1840_2,v100,z5,Soporte_final\WObj:=ADWob_2;
        MoveL Target_1850_2,v100,z5,Soporte_final\WObj:=ADWob_2;
        MoveL Target_1860_2,v100,z5,Soporte_final\WObj:=ADWob_2;
        MoveL Target_1870_2,v100,z5,Soporte_final\WObj:=ADWob_2;
        MoveL Target_1880_2,v100,z5,Soporte_final\WObj:=ADWob_2;
        MoveL Target_1890_2,v100,z5,Soporte_final\WObj:=ADWob_2;
        MoveL Target_1900_2,v100,z5,Soporte_final\WObj:=ADWob_2;
        MoveL Target_1910_2,v100,z5,Soporte_final\WObj:=ADWob_2;
        MoveL Target_1920_2,v100,z5,Soporte_final\WObj:=ADWob_2;
        MoveL Target_1930_2,v100,z5,Soporte_final\WObj:=ADWob_2;
        MoveL Target_1940_2,v100,z5,Soporte_final\WObj:=ADWob_2;
        MoveL Target_1950_2,v100,z5,Soporte_final\WObj:=ADWob_2;
        MoveL Target_1960_2,v100,z5,Soporte_final\WObj:=ADWob_2;
        MoveL Target_1970_2,v100,z5,Soporte_final\WObj:=ADWob_2;
        MoveL Target_1980_2,v100,z5,Soporte_final\WObj:=ADWob_2;
        MoveL Target_1990_2,v100,z5,Soporte_final\WObj:=ADWob_2;
        MoveL Target_2000_2,v100,z5,Soporte_final\WObj:=ADWob_2;
        MoveL Target_2010_2,v100,z5,Soporte_final\WObj:=ADWob_2;
        MoveL Target_2020_2,v100,z5,Soporte_final\WObj:=ADWob_2;
        MoveL Target_2030_2,v100,z5,Soporte_final\WObj:=ADWob_2;
        MoveL Target_2040_2,v100,z5,Soporte_final\WObj:=ADWob_2;
        MoveL Target_2050_2,v100,z5,Soporte_final\WObj:=ADWob_2;
        MoveL Target_2060_2,v100,z5,Soporte_final\WObj:=ADWob_2;
        MoveL Target_2070_2,v100,z5,Soporte_final\WObj:=ADWob_2;
        MoveL Target_2080_2,v100,z5,Soporte_final\WObj:=ADWob_2;
        MoveL Target_2090_2,v100,z5,Soporte_final\WObj:=ADWob_2;
        MoveL Target_2100_2,v100,z5,Soporte_final\WObj:=ADWob_2;
        MoveL Target_2110_2,v100,z5,Soporte_final\WObj:=ADWob_2;
        MoveL Target_2120_2,v100,z5,Soporte_final\WObj:=ADWob_2;
        MoveL Target_2130_2,v100,z5,Soporte_final\WObj:=ADWob_2;
        MoveL Target_2140_2,v100,z5,Soporte_final\WObj:=ADWob_2;
        MoveL Target_2150_2,v100,z5,Soporte_final\WObj:=ADWob_2;
        MoveL Target_2160_2,v100,z5,Soporte_final\WObj:=ADWob_2;
        MoveL Target_2170_2,v100,z5,Soporte_final\WObj:=ADWob_2;
        MoveL Target_2180_2,v100,z5,Soporte_final\WObj:=ADWob_2;
        MoveL Target_2190_2,v100,z5,Soporte_final\WObj:=ADWob_2;
        MoveL Target_2200_2,v100,z5,Soporte_final\WObj:=ADWob_2;
        MoveL Target_2210_2,v100,z5,Soporte_final\WObj:=ADWob_2;
        MoveL Target_2220_2,v100,z5,Soporte_final\WObj:=ADWob_2;
        MoveL Target_2230_2,v100,z5,Soporte_final\WObj:=ADWob_2;
        MoveL Target_2240_2,v100,z5,Soporte_final\WObj:=ADWob_2;
        MoveL Target_1380_2,v100,z5,Soporte_final\WObj:=ADWob_2; !une letra a ultima
        MoveL Target_1370_2,v100,z5,Soporte_final\WObj:=ADWob_2; !sube en z
        MoveL Target_2250_2,v100,z5,Soporte_final\WObj:=ADWob_2; !circulos de las cosas
        MoveL Target_2260_2,v100,z5,Soporte_final\WObj:=ADWob_2;  !baja en z
        MoveL Target_2270_2,v100,z5,Soporte_final\WObj:=ADWob_2;
        MoveL Target_2280_2,v100,z5,Soporte_final\WObj:=ADWob_2;
        MoveL Target_2290_2,v100,z5,Soporte_final\WObj:=ADWob_2;
        MoveL Target_2300_2,v100,z5,Soporte_final\WObj:=ADWob_2;
        MoveL Target_2310_2,v100,z5,Soporte_final\WObj:=ADWob_2;
        MoveL Target_2320_2,v100,z5,Soporte_final\WObj:=ADWob_2;
        MoveL Target_2340_2,v100,z5,Soporte_final\WObj:=ADWob_2;
        MoveL Target_2350_2,v100,z5,Soporte_final\WObj:=ADWob_2;
        MoveL Target_2360_2,v100,z5,Soporte_final\WObj:=ADWob_2;
        MoveL Target_2370_2,v100,z5,Soporte_final\WObj:=ADWob_2;
        MoveL Target_2380_2,v100,z5,Soporte_final\WObj:=ADWob_2;
        MoveL Target_2390_2,v100,z5,Soporte_final\WObj:=ADWob_2;
        MoveL Target_2400_2,v100,z5,Soporte_final\WObj:=ADWob_2;
        MoveL Target_2410_2,v100,z5,Soporte_final\WObj:=ADWob_2;
        MoveL Target_2420_2,v100,z5,Soporte_final\WObj:=ADWob_2;
        MoveL Target_2430_2,v100,z5,Soporte_final\WObj:=ADWob_2;
        MoveL Target_2440_2,v100,z5,Soporte_final\WObj:=ADWob_2;
        MoveL Target_2450_2,v100,z5,Soporte_final\WObj:=ADWob_2;
        MoveL Target_2460_2,v100,z5,Soporte_final\WObj:=ADWob_2;
        MoveL Target_2470_2,v100,z5,Soporte_final\WObj:=ADWob_2;
        MoveL Target_2260_2,v100,z5,Soporte_final\WObj:=ADWob_2; !cierra circulo de a
        MoveL Target_2250_2,v100,z5,Soporte_final\WObj:=ADWob_2; !sube en z
        MoveL Target_2330_2,v100,z5,Soporte_final\WObj:=ADWob_2; !llega arriba en d
        MoveL Target_2500_2,v100,z5,Soporte_final\WObj:=ADWob_2;
        MoveL Target_2510_2,v100,z5,Soporte_final\WObj:=ADWob_2;
        MoveL Target_2520_2,v100,z5,Soporte_final\WObj:=ADWob_2;
        MoveL Target_2530_2,v100,z5,Soporte_final\WObj:=ADWob_2;
        MoveL Target_2540_2,v100,z5,Soporte_final\WObj:=ADWob_2;
        MoveL Target_2550_2,v100,z5,Soporte_final\WObj:=ADWob_2;
        MoveL Target_2560_2,v100,z5,Soporte_final\WObj:=ADWob_2;
        MoveL Target_2570_2,v100,z5,Soporte_final\WObj:=ADWob_2;
        MoveL Target_2580_2,v100,z5,Soporte_final\WObj:=ADWob_2;
        MoveL Target_2590_2,v100,z5,Soporte_final\WObj:=ADWob_2;
        MoveL Target_2600_2,v100,z5,Soporte_final\WObj:=ADWob_2;
        MoveL Target_2610_2,v100,z5,Soporte_final\WObj:=ADWob_2;
        MoveL Target_2620_2,v100,z5,Soporte_final\WObj:=ADWob_2;
        MoveL Target_2630_2,v100,z5,Soporte_final\WObj:=ADWob_2;
        MoveL Target_2640_2,v100,z5,Soporte_final\WObj:=ADWob_2;
        MoveL Target_2650_2,v100,z5,Soporte_final\WObj:=ADWob_2;
        MoveL Target_2660_2,v100,z5,Soporte_final\WObj:=ADWob_2;
        MoveL Target_2670_2,v100,z5,Soporte_final\WObj:=ADWob_2;
        MoveL Target_2690_2,v100,z5,Soporte_final\WObj:=ADWob_2;
        MoveL Target_2700_2,v100,z5,Soporte_final\WObj:=ADWob_2;
        MoveL Target_2710_2,v100,z5,Soporte_final\WObj:=ADWob_2;
        MoveL Target_2720_2,v100,z5,Soporte_final\WObj:=ADWob_2;
        MoveL Target_2730_2,v100,z5,Soporte_final\WObj:=ADWob_2;
        MoveL Target_2740_2,v100,z5,Soporte_final\WObj:=ADWob_2;
        MoveL Target_2750_2,v100,z5,Soporte_final\WObj:=ADWob_2;
        MoveL Target_2500_2,v100,z5,Soporte_final\WObj:=ADWob_2;
        MoveL Target_2330_2,v100,z5,Soporte_final\WObj:=ADWob_2;
        MoveL Target_2760_2,v100,z5,Soporte_final\WObj:=ADWob_2;
        MoveL Target_2770_2,v100,z5,Soporte_final\WObj:=ADWob_2;
        MoveL Target_2780_2,v100,z5,Soporte_final\WObj:=ADWob_2;
        MoveL Target_2790_2,v100,z5,Soporte_final\WObj:=ADWob_2;
        MoveL Target_2800_2,v100,z5,Soporte_final\WObj:=ADWob_2;
        MoveL Target_2810_2,v100,z5,Soporte_final\WObj:=ADWob_2;
        MoveL Target_2820_2,v100,z5,Soporte_final\WObj:=ADWob_2;
        MoveL Target_2830_2,v100,z5,Soporte_final\WObj:=ADWob_2;
        MoveL Target_2840_2,v100,z5,Soporte_final\WObj:=ADWob_2;
        MoveL Target_2850_2,v100,z5,Soporte_final\WObj:=ADWob_2;
        MoveL Target_2860_2,v100,z5,Soporte_final\WObj:=ADWob_2;
        MoveL Target_2870_2,v100,z5,Soporte_final\WObj:=ADWob_2;
        MoveL Target_2880_2,v100,z5,Soporte_final\WObj:=ADWob_2;
        MoveL Target_2890_2,v100,z5,Soporte_final\WObj:=ADWob_2;
        MoveL Target_2900_2,v100,z5,Soporte_final\WObj:=ADWob_2;
        MoveL Target_2910_2,v100,z5,Soporte_final\WObj:=ADWob_2;
        MoveL Target_2770_2,v100,z5,Soporte_final\WObj:=ADWob_2;
        MoveL Target_2760_2,v100,z5,Soporte_final\WObj:=ADWob_2; ! queda arriba final.
        MoveJ Target_minihome_2,v100,z5,Soporte_final\WObj:=ADWob_2;
        MoveJ Target_minihome_2,v100,z5,Soporte_final\WObj:=ADWob_2;
        MoveL Target_2920_up_2,v100,z5,Soporte_final\WObj:=ADWob_2;
        MoveL Target_2920_2,v100,z5,Soporte_final\WObj:=ADWob_2;
        MoveL Target_2930_2,v100,z5,Soporte_final\WObj:=ADWob_2;
        MoveC Target_2940,Target_2950_2,v100,z5,Soporte_final\WObj:=ADWob_2;
        MoveL Target_2960_2,v100,z5,Soporte_final\WObj:=ADWob_2;
                MoveL Target_2920_2,v100,z5,Soporte_final\WObj:=ADWob_2;
        MoveL Target_2970_up_2,v100,z5,Soporte_final\WObj:=ADWob_2;
        MoveL Target_2970_2,v100,z5,Soporte_final\WObj:=ADWob_2;
        MoveL Target_2980_2,v100,z5,Soporte_final\WObj:=ADWob_2;
        MoveC Target_2990,Target_3000_2,v100,z5,Soporte_final\WObj:=ADWob_2;
        MoveL Target_3010_2,v100,z5,Soporte_final\WObj:=ADWob_2;
                MoveL Target_2970_2,v100,z5,Soporte_final\WObj:=ADWob_2;
        MoveL Target_3030_2_2,v100,z5,Soporte_final\WObj:=ADWob_2;
        MoveL Target_3030_2,v100,z5,Soporte_final\WObj:=ADWob_2;
        MoveL Target_3040_2,v100,z5,Soporte_final\WObj:=ADWob_2;
        MoveL Target_3050_2,v100,z5,Soporte_final\WObj:=ADWob_2;
        MoveL Target_3060_2,v100,z5,Soporte_final\WObj:=ADWob_2;
        MoveL Target_3070_2,v100,z5,Soporte_final\WObj:=ADWob_2;
        MoveL Target_3080_2,v100,z5,Soporte_final\WObj:=ADWob_2;
        MoveL Target_3090_2,v100,z5,Soporte_final\WObj:=ADWob_2;
        MoveL Target_3100_2,v100,z5,Soporte_final\WObj:=ADWob_2;
        MoveL Target_3110_2,v100,z5,Soporte_final\WObj:=ADWob_2;
        MoveL Target_3120_2,v100,z5,Soporte_final\WObj:=ADWob_2;
        MoveL Target_3130_2,v100,z5,Soporte_final\WObj:=ADWob_2;
        MoveL Target_3140_2,v100,z5,Soporte_final\WObj:=ADWob_2;
        MoveL Target_3150_2,v100,z5,Soporte_final\WObj:=ADWob_2;
        MoveL Target_3160_2,v100,z5,Soporte_final\WObj:=ADWob_2;
        MoveL Target_3170_2,v100,z5,Soporte_final\WObj:=ADWob_2;
        MoveL Target_3180_2,v100,z5,Soporte_final\WObj:=ADWob_2;
        MoveL Target_3190_2,v100,z5,Soporte_final\WObj:=ADWob_2;
        MoveL Target_3200_2,v100,z5,Soporte_final\WObj:=ADWob_2;
        MoveL Target_3210_2,v100,z5,Soporte_final\WObj:=ADWob_2;
        MoveL Target_3220_2,v100,z5,Soporte_final\WObj:=ADWob_2;
        MoveL Target_3230_2,v100,z5,Soporte_final\WObj:=ADWob_2;
        MoveL Target_3240_2,v100,z5,Soporte_final\WObj:=ADWob_2;
        MoveL Target_3250_2,v100,z5,Soporte_final\WObj:=ADWob_2;
        MoveL Target_3030_2,v100,z5,Soporte_final\WObj:=ADWob_2;
        MoveL Target_3260_2_2,v100,z5,Soporte_final\WObj:=ADWob_2;
        MoveL Target_3260_2,v100,z5,Soporte_final\WObj:=ADWob_2;
        MoveL Target_3270_2,v100,z5,Soporte_final\WObj:=ADWob_2;
        MoveL Target_3280_2,v100,z5,Soporte_final\WObj:=ADWob_2;
        MoveL Target_3290_2,v100,z5,Soporte_final\WObj:=ADWob_2;
        MoveL Target_3300_2,v100,z5,Soporte_final\WObj:=ADWob_2;
        MoveL Target_3310_2,v100,z5,Soporte_final\WObj:=ADWob_2;
        MoveL Target_3320_2,v100,z5,Soporte_final\WObj:=ADWob_2;
        MoveL Target_3330_2,v100,z5,Soporte_final\WObj:=ADWob_2;
        MoveL Target_3340_2,v100,z5,Soporte_final\WObj:=ADWob_2;
        MoveL Target_3260_2,v100,z5,Soporte_final\WObj:=ADWob_2;
        MoveL Target_3350_2_2,v100,z5,Soporte_final\WObj:=ADWob_2;
        MoveL Target_3350_2,v100,z5,Soporte_final\WObj:=ADWob_2;
        MoveL Target_3360_2,v100,z5,Soporte_final\WObj:=ADWob_2;
        MoveL Target_3370_2,v100,z5,Soporte_final\WObj:=ADWob_2;
        MoveL Target_3380_2,v100,z5,Soporte_final\WObj:=ADWob_2;
        MoveL Target_3390_2,v100,z5,Soporte_final\WObj:=ADWob_2;
        MoveL Target_3400_2,v100,z5,Soporte_final\WObj:=ADWob_2;
        MoveL Target_3410_2,v100,z5,Soporte_final\WObj:=ADWob_2;
        MoveL Target_3350_2,v100,z5,Soporte_final\WObj:=ADWob_2;
        MoveL Target_3420_2_2,v100,z5,Soporte_final\WObj:=ADWob_2;
        MoveL Target_3420_2,v100,z5,Soporte_final\WObj:=ADWob_2;
        MoveL Target_3430_2,v100,z5,Soporte_final\WObj:=ADWob_2;
        MoveL Target_3440_2,v100,z5,Soporte_final\WObj:=ADWob_2;
        MoveL Target_3450_2,v100,z5,Soporte_final\WObj:=ADWob_2;
        MoveL Target_3420_2,v100,z5,Soporte_final\WObj:=ADWob_2;
        MoveL Target_3460_2_2,v100,z5,Soporte_final\WObj:=ADWob_2;
        MoveL Target_3460_2,v100,z5,Soporte_final\WObj:=ADWob_2;
        MoveL Target_3470_2,v100,z5,Soporte_final\WObj:=ADWob_2;
        MoveL Target_3480_2,v100,z5,Soporte_final\WObj:=ADWob_2;
        MoveL Target_3490_2,v100,z5,Soporte_final\WObj:=ADWob_2;
        MoveL Target_3500_2,v100,z5,Soporte_final\WObj:=ADWob_2;
        MoveL Target_3510_2,v100,z5,Soporte_final\WObj:=ADWob_2;
                MoveL Target_3460_2,v100,z5,Soporte_final\WObj:=ADWob_2;
                MoveL Target_3520_2_2,v100,z5,Soporte_final\WObj:=ADWob_2;
                MoveL Target_3520_2,v100,z5,Soporte_final\WObj:=ADWob_2;
        MoveL Target_3530_2,v100,z5,Soporte_final\WObj:=ADWob_2;
        MoveL Target_3540_2,v100,z5,Soporte_final\WObj:=ADWob_2;
        MoveL Target_3550_2,v100,z5,Soporte_final\WObj:=ADWob_2;
        MoveL Target_3560_2,v100,z5,Soporte_final\WObj:=ADWob_2;
        MoveL Target_3570_2,v100,z5,Soporte_final\WObj:=ADWob_2;
        MoveL Target_3580_2,v100,z5,Soporte_final\WObj:=ADWob_2;
                MoveL Target_3590_2,v100,z5,Soporte_final\WObj:=ADWob_2;
                MoveL Target_3600_2,v100,z5,Soporte_final\WObj:=ADWob_2;
        MoveL Target_3610_2,v100,z5,Soporte_final\WObj:=ADWob_2;
        MoveL Target_3620_2,v100,z5,Soporte_final\WObj:=ADWob_2;
        MoveL Target_3630_2,v100,z5,Soporte_final\WObj:=ADWob_2;
        MoveL Target_3640_2,v100,z5,Soporte_final\WObj:=ADWob_2;
        MoveL Target_3650_2,v100,z5,Soporte_final\WObj:=ADWob_2;
        MoveL Target_3660_2,v100,z5,Soporte_final\WObj:=ADWob_2;
        MoveL Target_3520_2,v100,z5,Soporte_final\WObj:=ADWob_2;
                MoveL Target_3670_2_2,v100,z5,Soporte_final\WObj:=ADWob_2;
                MoveL Target_3670_2,v100,z5,Soporte_final\WObj:=ADWob_2;
                MoveL Target_3680_2,v100,z5,Soporte_final\WObj:=ADWob_2;
        MoveL Target_3690_2,v100,z5,Soporte_final\WObj:=ADWob_2;
        MoveL Target_3700_2,v100,z5,Soporte_final\WObj:=ADWob_2;
        MoveL Target_3710_2,v100,z5,Soporte_final\WObj:=ADWob_2;
        MoveL Target_3720_2,v100,z5,Soporte_final\WObj:=ADWob_2;
        MoveL Target_3730_2,v100,z5,Soporte_final\WObj:=ADWob_2;
        MoveL Target_3740_2,v100,z5,Soporte_final\WObj:=ADWob_2;
        MoveL Target_3670_2,v100,z5,Soporte_final\WObj:=ADWob_2;
        MoveJ Target_minihome_2,v100,z5,Soporte_final\WObj:=ADWob_2;
                MoveL Target_3750_2_2,v100,z5,Soporte_final\WObj:=ADWob_2;
        MoveL Target_3750_2,v100,z5,Soporte_final\WObj:=ADWob_2;
        MoveL Target_3760_2,v100,z5,Soporte_final\WObj:=ADWob_2;
        MoveL Target_3770_2,v100,z5,Soporte_final\WObj:=ADWob_2;
        MoveL Target_3780_2,v100,z5,Soporte_final\WObj:=ADWob_2;
        MoveL Target_3790_2,v100,z5,Soporte_final\WObj:=ADWob_2;
        MoveL Target_3800_2,v100,z5,Soporte_final\WObj:=ADWob_2;
        MoveL Target_3810_2,v100,z5,Soporte_final\WObj:=ADWob_2;
        MoveL Target_3820_2,v100,z5,Soporte_final\WObj:=ADWob_2;
        MoveL Target_3830_2,v100,z5,Soporte_final\WObj:=ADWob_2;
        MoveL Target_3840_2,v100,z5,Soporte_final\WObj:=ADWob_2;
        MoveL Target_3850_2,v100,z5,Soporte_final\WObj:=ADWob_2;
        MoveL Target_3860_2,v100,z5,Soporte_final\WObj:=ADWob_2;
        MoveL Target_3870_2,v100,z5,Soporte_final\WObj:=ADWob_2;
        MoveL Target_3880_2,v100,z5,Soporte_final\WObj:=ADWob_2;
        MoveL Target_3890_2,v100,z5,Soporte_final\WObj:=ADWob_2;
        MoveL Target_3900_2,v100,z5,Soporte_final\WObj:=ADWob_2;
                MoveL Target_3750_2,v100,z5,Soporte_final\WObj:=ADWob_2;
                MoveL Target_3910_2_2,v100,z5,Soporte_final\WObj:=ADWob_2;
        MoveL Target_3910_2,v100,z5,Soporte_final\WObj:=ADWob_2;
        MoveL Target_3920_2,v100,z5,Soporte_final\WObj:=ADWob_2;
        MoveL Target_3930_2,v100,z5,Soporte_final\WObj:=ADWob_2;
        MoveL Target_3940_2,v100,z5,Soporte_final\WObj:=ADWob_2;
        MoveL Target_3950_2,v100,z5,Soporte_final\WObj:=ADWob_2;
        MoveL Target_3960_2,v100,z5,Soporte_final\WObj:=ADWob_2;
                MoveL Target_3910_2,v100,z5,Soporte_final\WObj:=ADWob_2;
                MoveL Target_3970_2_2,v100,z5,Soporte_final\WObj:=ADWob_2;
        MoveL Target_3970_2,v100,z5,Soporte_final\WObj:=ADWob_2;
        MoveL Target_3980_2,v100,z5,Soporte_final\WObj:=ADWob_2;
        MoveL Target_3990_2,v100,z5,Soporte_final\WObj:=ADWob_2;
        MoveL Target_4000_2,v100,z5,Soporte_final\WObj:=ADWob_2;
                MoveL Target_3970_2,v100,z5,Soporte_final\WObj:=ADWob_2;
                MoveL Target_4010_2_2,v100,z5,Soporte_final\WObj:=ADWob_2;
        MoveL Target_4010_2,v100,z5,Soporte_final\WObj:=ADWob_2;
        MoveL Target_4020_2,v100,z5,Soporte_final\WObj:=ADWob_2;
        MoveL Target_4030_2,v100,z5,Soporte_final\WObj:=ADWob_2;
        MoveL Target_4040_2,v100,z5,Soporte_final\WObj:=ADWob_2;
        MoveL Target_4050_2,v100,z5,Soporte_final\WObj:=ADWob_2;
        MoveL Target_4060_2,v100,z5,Soporte_final\WObj:=ADWob_2;
        MoveL Target_4070_2,v100,z5,Soporte_final\WObj:=ADWob_2;
        MoveL Target_4080_2,v100,z5,Soporte_final\WObj:=ADWob_2;
        MoveL Target_4090_2,v100,z5,Soporte_final\WObj:=ADWob_2;
        MoveL Target_4100_2,v100,z5,Soporte_final\WObj:=ADWob_2;
        MoveL Target_4110_2,v100,z5,Soporte_final\WObj:=ADWob_2;
        MoveL Target_4120_2,v100,z5,Soporte_final\WObj:=ADWob_2;
        MoveL Target_4130_2,v100,z5,Soporte_final\WObj:=ADWob_2;
        MoveL Target_4010_2,v100,z5,Soporte_final\WObj:=ADWob_2;
        MoveL Target_minihome_2,v100,z5,Soporte_final\WObj:=ADWob_2;
    ENDPROC

ENDMODULE

--- Controller Data/IRB140_6_81/SYSPAR/EIO.cfg ---
EIO:CFG_1.0:6:1::
#
EIO_SIGNAL:

      -Name "Conveyor_INV" -SignalType "DO"

      -Name "DI_01" -SignalType "DI"

      -Name "DI_02" -SignalType "DI"

      -Name "DO_01" -SignalType "DO"

      -Name "DO_02" -SignalType "DO"
